LIN {X 0,Y 284.606,Z 589.036,A -85,B 0,C 180,E1 -17094.331,E2 -17094.331} C_VEL
LIN {X 0,Y 284.86,Z 589.002,A -85,B 0,C 180,E1 -17098.586,E2 -17098.586} C_VEL
LIN {X 0,Y 284.86,Z 588.997,A -85,B 0,C 180,E1 -17101.413,E2 -17101.413} C_VEL
LIN {X 0,Y 284.703,Z 589.017,A -85,B 0,C 180,E1 -17107.089,E2 -17107.089} C_VEL
LIN {X 0,Y 284.571,Z 589.036,A -85,B 0,C 180,E1 -17109.955,E2 -17109.955} C_VEL
LIN {X 0,Y 284.482,Z 589.046,A -85,B 0,C 180,E1 -17114.302,E2 -17114.302} C_VEL
LIN {X 0,Y 284.429,Z 589.048,A -85,B 0,C 180,E1 -17117.247,E2 -17117.247} C_VEL
LIN {X 0,Y 284.382,Z 589.061,A -85,B 0,C 180,E1 -17120.241,E2 -17120.241} C_VEL
LIN {X 0,Y 284.372,Z 589.06,A -85,B 0,C 180,E1 -17123.874,E2 -17123.874} C_VEL
LIN {X 0,Y 284.4,Z 589.052,A -85,B 0,C 180,E1 -17127.173,E2 -17127.173} C_VEL
LIN {X 0,Y 284.298,Z 589.069,A -85,B 0,C 180,E1 -17131.273,E2 -17131.273} C_VEL
LIN {X 0,Y 284.343,Z 589.063,A -85,B 0,C 180,E1 -17135.347,E2 -17135.347} C_VEL
LIN {X 0,Y 284.314,Z 589.069,A -85,B 0,C 180,E1 -17138.168,E2 -17138.168} C_VEL
LIN {X 0,Y 284.271,Z 589.074,A -85,B 0,C 180,E1 -17142.123,E2 -17142.123} C_VEL
LIN {X 0,Y 284.287,Z 589.069,A -85,B 0,C 180,E1 -17146.194,E2 -17146.194} C_VEL
LIN {X 0,Y 284.314,Z 589.068,A -85,B 0,C 180,E1 -17150.021,E2 -17150.021} C_VEL
LIN {X 0,Y 284.351,Z 589.061,A -85,B 0,C 180,E1 -17153.616,E2 -17153.616} C_VEL
LIN {X 0,Y 284.308,Z 589.067,A -85,B 0,C 180,E1 -17157.189,E2 -17157.189} C_VEL
LIN {X 0,Y 284.356,Z 589.065,A -85,B 0,C 180,E1 -17160.374,E2 -17160.374} C_VEL
LIN {X 0,Y 284.375,Z 589.058,A -85,B 0,C 180,E1 -17163.585,E2 -17163.585} C_VEL
LIN {X 0,Y 284.367,Z 589.063,A -85,B 0,C 180,E1 -17166.706,E2 -17166.706} C_VEL
LIN {X 0,Y 284.403,Z 589.057,A -85,B 0,C 180,E1 -17171.26,E2 -17171.26} C_VEL
LIN {X 0,Y 284.492,Z 589.045,A -85,B 0,C 180,E1 -17174.458,E2 -17174.458} C_VEL
LIN {X 0,Y 284.489,Z 589.047,A -85,B 0,C 180,E1 -17178.6,E2 -17178.6} C_VEL
LIN {X 0,Y 284.668,Z 589.024,A -85,B 0,C 180,E1 -17181.525,E2 -17181.525} C_VEL
LIN {X 0,Y 288.557,Z 601.326,A -85,B 0,C 180,E1 -17182.828,E2 -17182.828} C_VEL
LIN {X 0,Y 291.525,Z 612.433,A -85,B 0,C 180,E1 -17184.223,E2 -17184.223} C_VEL
LIN {X 0,Y 291.996,Z 614.209,A -85,B 0,C 180,E1 -17184.474,E2 -17184.474} C_VEL
LIN {X 0,Y 290.847,Z 625.708,A -85,B 0,C 180,E1 -17186.015,E2 -17186.015} C_VEL
LIN {X 0,Y 289.812,Z 634.995,A -85,B 0,C 180,E1 -17187.567,E2 -17187.567} C_VEL
LIN {X 0,Y 288.604,Z 643.761,A -85,B 0,C 180,E1 -17189.353,E2 -17189.353} C_VEL
LIN {X 0,Y 287.536,Z 651.804,A -85,B 0,C 180,E1 -17191.399,E2 -17191.399} C_VEL
LIN {X 0,Y 286.639,Z 658.483,A -85,B 0,C 180,E1 -17193.513,E2 -17193.513} C_VEL
LIN {X 0,Y 285.832,Z 663.856,A -85,B 0,C 180,E1 -17195.643,E2 -17195.643} C_VEL
LIN {X 0,Y 285.275,Z 668.057,A -85,B 0,C 180,E1 -17197.786,E2 -17197.786} C_VEL
LIN {X 0,Y 284.872,Z 671.215,A -85,B 0,C 180,E1 -17199.943,E2 -17199.943} C_VEL
LIN {X 0,Y 284.756,Z 672.789,A -85,B 0,C 180,E1 -17201.386,E2 -17201.386} C_VEL
LIN {X 0,Y 284.704,Z 673.91,A -85,B 0,C 180,E1 -17202.835,E2 -17202.835} C_VEL
LIN {X 0,Y 284.97,Z 674.965,A -85,B 0,C 180,E1 -17205.739,E2 -17205.739} C_VEL
LIN {X 0,Y 285.182,Z 674.889,A -85,B 0,C 180,E1 -17207.2,E2 -17207.2} C_VEL
LIN {X 0,Y 285.511,Z 674.378,A -85,B 0,C 180,E1 -17208.661,E2 -17208.661} C_VEL
LIN {X 0,Y 286.381,Z 672.543,A -85,B 0,C 180,E1 -17211.166,E2 -17211.166} C_VEL
LIN {X 0,Y 287.626,Z 669.263,A -85,B 0,C 180,E1 -17213.775,E2 -17213.775} C_VEL
LIN {X 0,Y 288.934,Z 665.274,A -85,B 0,C 180,E1 -17215.964,E2 -17215.964} C_VEL
LIN {X 0,Y 290.739,Z 659.013,A -85,B 0,C 180,E1 -17218.515,E2 -17218.515} C_VEL
LIN {X 0,Y 292.655,Z 652.073,A -85,B 0,C 180,E1 -17220.683,E2 -17220.683} C_VEL
LIN {X 0,Y 294.442,Z 644.856,A -85,B 0,C 180,E1 -17222.481,E2 -17222.481} C_VEL
LIN {X 0,Y 296.435,Z 635.72,A -85,B 0,C 180,E1 -17224.316,E2 -17224.316} C_VEL
LIN {X 0,Y 298.194,Z 626.062,A -85,B 0,C 180,E1 -17225.889,E2 -17225.889} C_VEL
LIN {X 0,Y 295.848,Z 617.051,A -85,B 0,C 180,E1 -17227.55,E2 -17227.55} C_VEL
LIN {X 0,Y 291.54,Z 610.398,A -85,B 0,C 180,E1 -17228.962,E2 -17228.962} C_VEL
LIN {X 0,Y 287.015,Z 604.55,A -85,B 0,C 180,E1 -17230.228,E2 -17230.228} C_VEL
LIN {X 0,Y 286.747,Z 603.732,A -85,B 0,C 180,E1 -17230.381,E2 -17230.381} C_VEL
LIN {X 0,Y 286.527,Z 609.898,A -85,B 0,C 180,E1 -17233.374,E2 -17233.374} C_VEL
LIN {X 0,Y 285.989,Z 617.64,A -85,B 0,C 180,E1 -17237.095,E2 -17237.095} C_VEL
LIN {X 0,Y 285.473,Z 626.048,A -85,B 0,C 180,E1 -17241.114,E2 -17241.114} C_VEL
LIN {X 0,Y 285.15,Z 632.582,A -85,B 0,C 180,E1 -17244.221,E2 -17244.221} C_VEL
LIN {X 0,Y 287.62,Z 646.522,A -85,B 0,C 180,E1 -17245.077,E2 -17245.077} C_VEL
LIN {X 0,Y 289.828,Z 659.569,A -85,B 0,C 180,E1 -17246.148,E2 -17246.148} C_VEL
LIN {X 0,Y 290.365,Z 664.219,A -85,B 0,C 180,E1 -17246.59,E2 -17246.59} C_VEL
LIN {X 0,Y 289.25,Z 676.311,A -85,B 0,C 180,E1 -17247.822,E2 -17247.822} C_VEL
LIN {X 0,Y 287.885,Z 688.211,A -85,B 0,C 180,E1 -17249.363,E2 -17249.363} C_VEL
LIN {X 0,Y 286.677,Z 698.653,A -85,B 0,C 180,E1 -17251.042,E2 -17251.042} C_VEL
LIN {X 0,Y 285.548,Z 708.096,A -85,B 0,C 180,E1 -17252.915,E2 -17252.915} C_VEL
LIN {X 0,Y 284.575,Z 715.877,A -85,B 0,C 180,E1 -17254.786,E2 -17254.786} C_VEL
LIN {X 0,Y 283.779,Z 723.483,A -85,B 0,C 180,E1 -17257.042,E2 -17257.042} C_VEL
LIN {X 0,Y 283.086,Z 730.338,A -85,B 0,C 180,E1 -17259.662,E2 -17259.662} C_VEL
LIN {X 0,Y 282.716,Z 734.782,A -85,B 0,C 180,E1 -17261.897,E2 -17261.897} C_VEL
LIN {X 0,Y 282.461,Z 738.031,A -85,B 0,C 180,E1 -17264.116,E2 -17264.116} C_VEL
LIN {X 0,Y 282.44,Z 739.964,A -85,B 0,C 180,E1 -17266.028,E2 -17266.028} C_VEL
LIN {X 0,Y 282.528,Z 741.392,A -85,B 0,C 180,E1 -17268.522,E2 -17268.522} C_VEL
LIN {X 0,Y 282.699,Z 741.622,A -85,B 0,C 180,E1 -17269.979,E2 -17269.979} C_VEL
LIN {X 0,Y 283.343,Z 740.915,A -85,B 0,C 180,E1 -17272.804,E2 -17272.804} C_VEL
LIN {X 0,Y 283.79,Z 739.87,A -85,B 0,C 180,E1 -17274.316,E2 -17274.316} C_VEL
LIN {X 0,Y 284.213,Z 738.56,A -85,B 0,C 180,E1 -17275.642,E2 -17275.642} C_VEL
LIN {X 0,Y 284.048,Z 737.349,A -85,B 0,C 180,E1 -17276.809,E2 -17276.809} C_VEL
LIN {X 0,Y 282.237,Z 735.003,A -85,B 0,C 180,E1 -17278.726,E2 -17278.726} C_VEL
LIN {X 0,Y 280.85,Z 732.632,A -85,B 0,C 180,E1 -17280.244,E2 -17280.244} C_VEL
LIN {X 0,Y 280.68,Z 730.45,A -85,B 0,C 180,E1 -17281.364,E2 -17281.364} C_VEL
LIN {X 0,Y 280.899,Z 729.624,A -85,B 0,C 180,E1 -17281.727,E2 -17281.727} C_VEL
LIN {X 0,Y 282.965,Z 723.832,A -85,B 0,C 180,E1 -17283.917,E2 -17283.917} C_VEL
LIN {X 0,Y 285.304,Z 716.83,A -85,B 0,C 180,E1 -17286.01,E2 -17286.01} C_VEL
LIN {X 0,Y 288.012,Z 708.164,A -85,B 0,C 180,E1 -17288.066,E2 -17288.066} C_VEL
LIN {X 0,Y 290.524,Z 699.534,A -85,B 0,C 180,E1 -17289.75,E2 -17289.75} C_VEL
LIN {X 0,Y 293.371,Z 688.781,A -85,B 0,C 180,E1 -17291.434,E2 -17291.434} C_VEL
LIN {X 0,Y 295.827,Z 677.662,A -85,B 0,C 180,E1 -17292.845,E2 -17292.845} C_VEL
LIN {X 0,Y 294.677,Z 667.632,A -85,B 0,C 180,E1 -17294.47,E2 -17294.47} C_VEL
LIN {X 0,Y 292.135,Z 657.124,A -85,B 0,C 180,E1 -17296.234,E2 -17296.234} C_VEL
LIN {X 0,Y 288.644,Z 647.19,A -85,B 0,C 180,E1 -17298.026,E2 -17298.026} C_VEL
LIN {X 0,Y 286.586,Z 642.357,A -85,B 0,C 180,E1 -17298.985,E2 -17298.985} C_VEL
LIN {X 0,Y 285.531,Z 639.392,A -85,B 0,C 180,E1 -17299.548,E2 -17299.548} C_VEL
LIN {X 0,Y 287.353,Z 632.653,A -85,B 0,C 180,E1 -17303.801,E2 -17303.801} C_VEL
LIN {X 0,Y 288.082,Z 629.504,A -85,B 0,C 180,E1 -17306.049,E2 -17306.049} C_VEL
LIN {X 0,Y 288.296,Z 626.554,A -85,B 0,C 180,E1 -17308.65,E2 -17308.65} C_VEL
LIN {X 0,Y 288.285,Z 624.039,A -85,B 0,C 180,E1 -17311.436,E2 -17311.436} C_VEL
LIN {X 0,Y 288.31,Z 622.174,A -85,B 0,C 180,E1 -17314.102,E2 -17314.102} C_VEL
LIN {X 0,Y 288.543,Z 620.675,A -85,B 0,C 180,E1 -17317.512,E2 -17317.512} C_VEL
LIN {X 0,Y 288.683,Z 620.382,A -85,B 0,C 180,E1 -17319.27,E2 -17319.27} C_VEL
LIN {X 0,Y 288.734,Z 620.549,A -85,B 0,C 180,E1 -17321.087,E2 -17321.087} C_VEL
LIN {X 0,Y 288.549,Z 621.433,A -85,B 0,C 180,E1 -17323.058,E2 -17323.058} C_VEL
LIN {X 0,Y 288.243,Z 623.559,A -85,B 0,C 180,E1 -17325.684,E2 -17325.684} C_VEL
LIN {X 0,Y 288.344,Z 627.834,A -85,B 0,C 180,E1 -17329.077,E2 -17329.077} C_VEL
LIN {X 0,Y 288.366,Z 629.026,A -85,B 0,C 180,E1 -17329.796,E2 -17329.796} C_VEL
LIN {X 0,Y 287.752,Z 633.355,A -85,B 0,C 180,E1 -17331.717,E2 -17331.717} C_VEL
LIN {X 0,Y 286.85,Z 639.765,A -85,B 0,C 180,E1 -17333.986,E2 -17333.986} C_VEL
LIN {X 0,Y 286.34,Z 648.27,A -85,B 0,C 180,E1 -17336.565,E2 -17336.565} C_VEL
LIN {X 0,Y 286.351,Z 652.539,A -85,B 0,C 180,E1 -17337.652,E2 -17337.652} C_VEL
LIN {X 0,Y 289.68,Z 665.175,A -85,B 0,C 180,E1 -17339.394,E2 -17339.394} C_VEL
LIN {X 0,Y 291.628,Z 675.536,A -85,B 0,C 180,E1 -17340.711,E2 -17340.711} C_VEL
LIN {X 0,Y 292.656,Z 687.693,A -85,B 0,C 180,E1 -17342.173,E2 -17342.173} C_VEL
LIN {X 0,Y 292.149,Z 698.271,A -85,B 0,C 180,E1 -17343.413,E2 -17343.413} C_VEL
LIN {X 0,Y 290.389,Z 710.468,A -85,B 0,C 180,E1 -17344.944,E2 -17344.944} C_VEL
LIN {X 0,Y 288.295,Z 721.832,A -85,B 0,C 180,E1 -17346.665,E2 -17346.665} C_VEL
LIN {X 0,Y 285.663,Z 731.527,A -85,B 0,C 180,E1 -17348.345,E2 -17348.345} C_VEL
LIN {X 0,Y 283.312,Z 739.677,A -85,B 0,C 180,E1 -17350.058,E2 -17350.058} C_VEL
LIN {X 0,Y 280.506,Z 749.053,A -85,B 0,C 180,E1 -17352.504,E2 -17352.504} C_VEL
LIN {X 0,Y 278.866,Z 755.583,A -85,B 0,C 180,E1 -17354.657,E2 -17354.657} C_VEL
LIN {X 0,Y 277.3,Z 760.909,A -85,B 0,C 180,E1 -17356.816,E2 -17356.816} C_VEL
LIN {X 0,Y 276.397,Z 765.123,A -85,B 0,C 180,E1 -17359.008,E2 -17359.008} C_VEL
LIN {X 0,Y 275.824,Z 768.335,A -85,B 0,C 180,E1 -17361.208,E2 -17361.208} C_VEL
LIN {X 0,Y 275.613,Z 769.942,A -85,B 0,C 180,E1 -17362.676,E2 -17362.676} C_VEL
LIN {X 0,Y 275.476,Z 771.938,A -85,B 0,C 180,E1 -17365.612,E2 -17365.612} C_VEL
LIN {X 0,Y 275.507,Z 772.333,A -85,B 0,C 180,E1 -17367.077,E2 -17367.077} C_VEL
LIN {X 0,Y 275.887,Z 771.819,A -85,B 0,C 180,E1 -17370.001,E2 -17370.001} C_VEL
LIN {X 0,Y 275.746,Z 770.912,A -85,B 0,C 180,E1 -17371.462,E2 -17371.462} C_VEL
LIN {X 0,Y 275.594,Z 769.545,A -85,B 0,C 180,E1 -17372.925,E2 -17372.925} C_VEL
LIN {X 0,Y 275.671,Z 766.636,A -85,B 0,C 180,E1 -17375.121,E2 -17375.121} C_VEL
LIN {X 0,Y 275.725,Z 762.583,A -85,B 0,C 180,E1 -17377.323,E2 -17377.323} C_VEL
LIN {X 0,Y 276.04,Z 756.286,A -85,B 0,C 180,E1 -17379.897,E2 -17379.897} C_VEL
LIN {X 0,Y 276.598,Z 749.373,A -85,B 0,C 180,E1 -17382.101,E2 -17382.101} C_VEL
LIN {X 0,Y 277.519,Z 740.696,A -85,B 0,C 180,E1 -17384.296,E2 -17384.296} C_VEL
LIN {X 0,Y 278.308,Z 733.752,A -85,B 0,C 180,E1 -17385.753,E2 -17385.753} C_VEL
LIN {X 0,Y 279.563,Z 723.375,A -85,B 0,C 180,E1 -17387.559,E2 -17387.559} C_VEL
LIN {X 0,Y 280.95,Z 711.747,A -85,B 0,C 180,E1 -17389.168,E2 -17389.168} C_VEL
LIN {X 0,Y 281.033,Z 701.802,A -85,B 0,C 180,E1 -17390.304,E2 -17390.304} C_VEL
LIN {X 0,Y 280.708,Z 689.594,A -85,B 0,C 180,E1 -17391.437,E2 -17391.437} C_VEL
LIN {X 0,Y 279.865,Z 675.724,A -85,B 0,C 180,E1 -17392.421,E2 -17392.421} C_VEL
LIN {X 0,Y 278.595,Z 659.43,A -85,B 0,C 180,E1 -17393.609,E2 -17393.609} C_VEL
LIN {X 0,Y 277.646,Z 651.097,A -85,B 0,C 180,E1 -17394.076,E2 -17394.076} C_VEL
LIN {X 0,Y 277.221,Z 642.295,A -85,B 0,C 180,E1 -17395.156,E2 -17395.156} C_VEL
LIN {X 0,Y 278.337,Z 631.986,A -85,B 0,C 180,E1 -17399.498,E2 -17399.498} C_VEL
LIN {X 0,Y 279.78,Z 621.349,A -85,B 0,C 180,E1 -17404.008,E2 -17404.008} C_VEL
LIN {X 0,Y 281.164,Z 612.603,A -85,B 0,C 180,E1 -17407.765,E2 -17407.765} C_VEL
LIN {X 0,Y 281.019,Z 609.529,A -85,B 0,C 180,E1 -17409.169,E2 -17409.169} C_VEL
LIN {X 0,Y 279.688,Z 602.149,A -85,B 0,C 180,E1 -17412.724,E2 -17412.724} C_VEL
LIN {X 0,Y 277.98,Z 593.465,A -85,B 0,C 180,E1 -17417.156,E2 -17417.156} C_VEL
LIN {X 0,Y 277.252,Z 589.953,A -85,B 0,C 180,E1 -17419.092,E2 -17419.092} C_VEL
LIN {X 0,Y 277.287,Z 589.951,A -85,B 0,C 180,E1 -17422.533,E2 -17422.533} C_VEL
LIN {X 0,Y 277.26,Z 589.953,A -85,B 0,C 180,E1 -17426.105,E2 -17426.105} C_VEL
LIN {X 0,Y 277.267,Z 589.947,A -85,B 0,C 180,E1 -17429.539,E2 -17429.539} C_VEL
LIN {X 0,Y 277.363,Z 589.934,A -85,B 0,C 180,E1 -17432.864,E2 -17432.864} C_VEL
LIN {X 0,Y 277.334,Z 589.94,A -85,B 0,C 180,E1 -17436.079,E2 -17436.079} C_VEL
LIN {X 0,Y 277.35,Z 589.937,A -85,B 0,C 180,E1 -17440.766,E2 -17440.766} C_VEL
LIN {X 0,Y 277.44,Z 589.925,A -85,B 0,C 180,E1 -17445.326,E2 -17445.326} C_VEL
LIN {X 0,Y 277.512,Z 589.916,A -85,B 0,C 180,E1 -17449.788,E2 -17449.788} C_VEL
LIN {X 0,Y 277.659,Z 589.898,A -85,B 0,C 180,E1 -17452.729,E2 -17452.729} C_VEL
LIN {X 0,Y 277.826,Z 589.879,A -85,B 0,C 180,E1 -17458.55,E2 -17458.55} C_VEL
LIN {X 0,Y 277.826,Z 589.874,A -85,B 0,C 180,E1 -17461.449,E2 -17461.449} C_VEL
LIN {X 0,Y 277.658,Z 589.894,A -85,B 0,C 180,E1 -17467.27,E2 -17467.27} C_VEL
LIN {X 0,Y 277.511,Z 589.917,A -85,B 0,C 180,E1 -17470.211,E2 -17470.211} C_VEL
LIN {X 0,Y 277.432,Z 589.92,A -85,B 0,C 180,E1 -17474.674,E2 -17474.674} C_VEL
LIN {X 0,Y 277.349,Z 589.934,A -85,B 0,C 180,E1 -17479.233,E2 -17479.233} C_VEL
LIN {X 0,Y 277.323,Z 589.94,A -85,B 0,C 180,E1 -17484.169,E2 -17484.169} C_VEL
LIN {X 0,Y 277.329,Z 589.932,A -85,B 0,C 180,E1 -17487.504,E2 -17487.504} C_VEL
LIN {X 0,Y 277.275,Z 589.948,A -85,B 0,C 180,E1 -17490.48,E2 -17490.48} C_VEL
LIN {X 0,Y 277.25,Z 589.947,A -85,B 0,C 180,E1 -17493.895,E2 -17493.895} C_VEL
LIN {X 0,Y 277.27,Z 589.944,A -85,B 0,C 180,E1 -17497.468,E2 -17497.468} C_VEL
LIN {X 0,Y 277.212,Z 589.952,A -85,B 0,C 180,E1 -17501.235,E2 -17501.235} C_VEL
LIN {X 0,Y 277.224,Z 589.946,A -85,B 0,C 180,E1 -17505.221,E2 -17505.221} C_VEL
LIN {X 0,Y 277.228,Z 589.952,A -85,B 0,C 180,E1 -17508.765,E2 -17508.765} C_VEL
LIN {X 0,Y 277.283,Z 589.943,A -85,B 0,C 180,E1 -17512.532,E2 -17512.532} C_VEL
LIN {X 0,Y 277.255,Z 589.948,A -85,B 0,C 180,E1 -17516.104,E2 -17516.104} C_VEL
LIN {X 0,Y 277.262,Z 589.945,A -85,B 0,C 180,E1 -17519.537,E2 -17519.537} C_VEL
LIN {X 0,Y 277.356,Z 589.934,A -85,B 0,C 180,E1 -17522.863,E2 -17522.863} C_VEL
LIN {X 0,Y 277.329,Z 589.939,A -85,B 0,C 180,E1 -17526.078,E2 -17526.078} C_VEL
LIN {X 0,Y 277.345,Z 589.939,A -85,B 0,C 180,E1 -17530.765,E2 -17530.765} C_VEL
LIN {X 0,Y 277.435,Z 589.924,A -85,B 0,C 180,E1 -17535.325,E2 -17535.325} C_VEL
LIN {X 0,Y 277.507,Z 589.917,A -85,B 0,C 180,E1 -17539.787,E2 -17539.787} C_VEL
LIN {X 0,Y 277.617,Z 589.902,A -85,B 0,C 180,E1 -17541.053,E2 -17541.053} C_VEL
LIN {X 0,Y 281.357,Z 601.323,A -85,B 0,C 180,E1 -17542.283,E2 -17542.283} C_VEL
LIN {X 0,Y 284.209,Z 612.288,A -85,B 0,C 180,E1 -17543.672,E2 -17543.672} C_VEL
LIN {X 0,Y 285.038,Z 615.32,A -85,B 0,C 180,E1 -17544.107,E2 -17544.107} C_VEL
LIN {X 0,Y 284.246,Z 624.779,A -85,B 0,C 180,E1 -17545.39,E2 -17545.39} C_VEL
LIN {X 0,Y 283.02,Z 635.357,A -85,B 0,C 180,E1 -17547.152,E2 -17547.152} C_VEL
LIN {X 0,Y 281.727,Z 644.666,A -85,B 0,C 180,E1 -17549.076,E2 -17549.076} C_VEL
LIN {X 0,Y 280.649,Z 652.285,A -85,B 0,C 180,E1 -17551.039,E2 -17551.039} C_VEL
LIN {X 0,Y 279.701,Z 659.158,A -85,B 0,C 180,E1 -17553.24,E2 -17553.24} C_VEL
LIN {X 0,Y 278.75,Z 665.41,A -85,B 0,C 180,E1 -17555.787,E2 -17555.787} C_VEL
LIN {X 0,Y 278.187,Z 669.492,A -85,B 0,C 180,E1 -17557.986,E2 -17557.986} C_VEL
LIN {X 0,Y 277.805,Z 672.538,A -85,B 0,C 180,E1 -17560.199,E2 -17560.199} C_VEL
LIN {X 0,Y 277.702,Z 674.009,A -85,B 0,C 180,E1 -17561.679,E2 -17561.679} C_VEL
LIN {X 0,Y 277.778,Z 675.743,A -85,B 0,C 180,E1 -17564.654,E2 -17564.654} C_VEL
LIN {X 0,Y 278.023,Z 676.005,A -85,B 0,C 180,E1 -17566.143,E2 -17566.143} C_VEL
LIN {X 0,Y 278.26,Z 675.84,A -85,B 0,C 180,E1 -17567.641,E2 -17567.641} C_VEL
LIN {X 0,Y 278.625,Z 675.278,A -85,B 0,C 180,E1 -17569.14,E2 -17569.14} C_VEL
LIN {X 0,Y 279.528,Z 673.5,A -85,B 0,C 180,E1 -17571.525,E2 -17571.525} C_VEL
LIN {X 0,Y 280.932,Z 669.885,A -85,B 0,C 180,E1 -17574.378,E2 -17574.378} C_VEL
LIN {X 0,Y 282.345,Z 665.765,A -85,B 0,C 180,E1 -17576.617,E2 -17576.617} C_VEL
LIN {X 0,Y 283.998,Z 660.378,A -85,B 0,C 180,E1 -17578.851,E2 -17578.851} C_VEL
LIN {X 0,Y 285.99,Z 653.521,A -85,B 0,C 180,E1 -17581.066,E2 -17581.066} C_VEL
LIN {X 0,Y 287.84,Z 646.411,A -85,B 0,C 180,E1 -17582.904,E2 -17582.904} C_VEL
LIN {X 0,Y 290.079,Z 636.717,A -85,B 0,C 180,E1 -17584.903,E2 -17584.903} C_VEL
LIN {X 0,Y 291.669,Z 628.681,A -85,B 0,C 180,E1 -17586.255,E2 -17586.255} C_VEL
LIN {X 0,Y 290.789,Z 623.926,A -85,B 0,C 180,E1 -17587.171,E2 -17587.171} C_VEL
LIN {X 0,Y 289.625,Z 620.101,A -85,B 0,C 180,E1 -17587.916,E2 -17587.916} C_VEL
LIN {X 0,Y 283.77,Z 611.791,A -85,B 0,C 180,E1 -17589.848,E2 -17589.848} C_VEL
LIN {X 0,Y 281.937,Z 609.423,A -85,B 0,C 180,E1 -17590.398,E2 -17590.398} C_VEL
LIN {X 0,Y 280.676,Z 608.353,A -85,B 0,C 180,E1 -17590.705,E2 -17590.705} C_VEL
LIN {X 0,Y 279.77,Z 606.539,A -85,B 0,C 180,E1 -17591.053,E2 -17591.053} C_VEL
LIN {X 0,Y 279.341,Z 614.142,A -85,B 0,C 180,E1 -17594.783,E2 -17594.783} C_VEL
LIN {X 0,Y 278.695,Z 623.179,A -85,B 0,C 180,E1 -17599.156,E2 -17599.156} C_VEL
LIN {X 0,Y 278.195,Z 631.942,A -85,B 0,C 180,E1 -17603.384,E2 -17603.384} C_VEL
LIN {X 0,Y 278.193,Z 633.111,A -85,B 0,C 180,E1 -17603.877,E2 -17603.877} C_VEL
LIN {X 0,Y 280.679,Z 647.191,A -85,B 0,C 180,E1 -17604.772,E2 -17604.772} C_VEL
LIN {X 0,Y 283,Z 661.237,A -85,B 0,C 180,E1 -17605.974,E2 -17605.974} C_VEL
LIN {X 0,Y 283.378,Z 665.151,A -85,B 0,C 180,E1 -17606.362,E2 -17606.362} C_VEL
LIN {X 0,Y 282.29,Z 676.434,A -85,B 0,C 180,E1 -17607.543,E2 -17607.543} C_VEL
LIN {X 0,Y 280.872,Z 688.513,A -85,B 0,C 180,E1 -17609.14,E2 -17609.14} C_VEL
LIN {X 0,Y 279.66,Z 698.989,A -85,B 0,C 180,E1 -17610.863,E2 -17610.863} C_VEL
LIN {X 0,Y 278.395,Z 709.305,A -85,B 0,C 180,E1 -17612.974,E2 -17612.974} C_VEL
LIN {X 0,Y 277.403,Z 717.108,A -85,B 0,C 180,E1 -17614.931,E2 -17614.931} C_VEL
LIN {X 0,Y 276.639,Z 724.416,A -85,B 0,C 180,E1 -17617.206,E2 -17617.206} C_VEL
LIN {X 0,Y 276.094,Z 729.425,A -85,B 0,C 180,E1 -17619.123,E2 -17619.123} C_VEL
LIN {X 0,Y 275.676,Z 734.164,A -85,B 0,C 180,E1 -17621.418,E2 -17621.418} C_VEL
LIN {X 0,Y 275.389,Z 737.699,A -85,B 0,C 180,E1 -17623.697,E2 -17623.697} C_VEL
LIN {X 0,Y 275.34,Z 740.106,A -85,B 0,C 180,E1 -17625.909,E2 -17625.909} C_VEL
LIN {X 0,Y 275.43,Z 741.605,A -85,B 0,C 180,E1 -17628.222,E2 -17628.222} C_VEL
LIN {X 0,Y 275.579,Z 742.047,A -85,B 0,C 180,E1 -17629.717,E2 -17629.717} C_VEL
LIN {X 0,Y 275.84,Z 742.055,A -85,B 0,C 180,E1 -17631.207,E2 -17631.207} C_VEL
LIN {X 0,Y 276.262,Z 741.57,A -85,B 0,C 180,E1 -17632.799,E2 -17632.799} C_VEL
LIN {X 0,Y 277.151,Z 739.605,A -85,B 0,C 180,E1 -17635.638,E2 -17635.638} C_VEL
LIN {X 0,Y 278.187,Z 736.982,A -85,B 0,C 180,E1 -17637.829,E2 -17637.829} C_VEL
LIN {X 0,Y 279.584,Z 733.346,A -85,B 0,C 180,E1 -17640.001,E2 -17640.001} C_VEL
LIN {X 0,Y 280.899,Z 729.624,A -85,B 0,C 180,E1 -17641.727,E2 -17641.727} C_VEL
LIN {X 0,Y 281.22,Z 727.146,A -85,B 0,C 180,E1 -17642.818,E2 -17642.818} C_VEL
LIN {X 0,Y 280.234,Z 722.98,A -85,B 0,C 180,E1 -17644.645,E2 -17644.645} C_VEL
LIN {X 0,Y 279.421,Z 718.315,A -85,B 0,C 180,E1 -17646.423,E2 -17646.423} C_VEL
LIN {X 0,Y 279.987,Z 714.995,A -85,B 0,C 180,E1 -17647.416,E2 -17647.416} C_VEL
LIN {X 0,Y 282.736,Z 706.842,A -85,B 0,C 180,E1 -17649.299,E2 -17649.299} C_VEL
LIN {X 0,Y 285.773,Z 696.756,A -85,B 0,C 180,E1 -17651.168,E2 -17651.168} C_VEL
LIN {X 0,Y 288.783,Z 685.636,A -85,B 0,C 180,E1 -17652.831,E2 -17652.831} C_VEL
LIN {X 0,Y 290.04,Z 680.443,A -85,B 0,C 180,E1 -17653.488,E2 -17653.488} C_VEL
LIN {X 0,Y 289.609,Z 673.403,A -85,B 0,C 180,E1 -17654.675,E2 -17654.675} C_VEL
LIN {X 0,Y 287.785,Z 663.263,A -85,B 0,C 180,E1 -17656.476,E2 -17656.476} C_VEL
LIN {X 0,Y 284.849,Z 653.325,A -85,B 0,C 180,E1 -17658.363,E2 -17658.363} C_VEL
LIN {X 0,Y 281.173,Z 643.852,A -85,B 0,C 180,E1 -17660.34,E2 -17660.34} C_VEL
LIN {X 0,Y 279.742,Z 640.057,A -85,B 0,C 180,E1 -17661.202,E2 -17661.202} C_VEL
LIN {X 0,Y 281.22,Z 635.336,A -85,B 0,C 180,E1 -17664.353,E2 -17664.353} C_VEL
LIN {X 0,Y 281.957,Z 632.366,A -85,B 0,C 180,E1 -17666.659,E2 -17666.659} C_VEL
LIN {X 0,Y 282.19,Z 629.601,A -85,B 0,C 180,E1 -17669.349,E2 -17669.349} C_VEL
LIN {X 0,Y 282.302,Z 627.32,A -85,B 0,C 180,E1 -17672.177,E2 -17672.177} C_VEL
LIN {X 0,Y 282.456,Z 625.761,A -85,B 0,C 180,E1 -17674.91,E2 -17674.91} C_VEL
LIN {X 0,Y 282.727,Z 624.862,A -85,B 0,C 180,E1 -17677.305,E2 -17677.305} C_VEL
LIN {X 0,Y 282.969,Z 624.61,A -85,B 0,C 180,E1 -17679.655,E2 -17679.655} C_VEL
LIN {X 0,Y 282.945,Z 625.292,A -85,B 0,C 180,E1 -17682.118,E2 -17682.118} C_VEL
LIN {X 0,Y 282.746,Z 626.648,A -85,B 0,C 180,E1 -17684.106,E2 -17684.106} C_VEL
LIN {X 0,Y 282.681,Z 629.477,A -85,B 0,C 180,E1 -17686.868,E2 -17686.868} C_VEL
LIN {X 0,Y 282.836,Z 632.31,A -85,B 0,C 180,E1 -17688.958,E2 -17688.958} C_VEL
LIN {X 0,Y 282.542,Z 635.249,A -85,B 0,C 180,E1 -17690.453,E2 -17690.453} C_VEL
LIN {X 0,Y 281.567,Z 641.182,A -85,B 0,C 180,E1 -17692.753,E2 -17692.753} C_VEL
LIN {X 0,Y 280.724,Z 650.383,A -85,B 0,C 180,E1 -17695.707,E2 -17695.707} C_VEL
LIN {X 0,Y 280.726,Z 652.091,A -85,B 0,C 180,E1 -17696.127,E2 -17696.127} C_VEL
LIN {X 0,Y 283.994,Z 664.357,A -85,B 0,C 180,E1 -17698.025,E2 -17698.025} C_VEL
LIN {X 0,Y 286.302,Z 677.17,A -85,B 0,C 180,E1 -17699.782,E2 -17699.782} C_VEL
LIN {X 0,Y 287.029,Z 689.116,A -85,B 0,C 180,E1 -17701.324,E2 -17701.324} C_VEL
LIN {X 0,Y 286.589,Z 697.866,A -85,B 0,C 180,E1 -17702.414,E2 -17702.414} C_VEL
LIN {X 0,Y 284.644,Z 710.053,A -85,B 0,C 180,E1 -17704.009,E2 -17704.009} C_VEL
LIN {X 0,Y 282.211,Z 722.401,A -85,B 0,C 180,E1 -17705.935,E2 -17705.935} C_VEL
LIN {X 0,Y 279.159,Z 732.656,A -85,B 0,C 180,E1 -17707.814,E2 -17707.814} C_VEL
LIN {X 0,Y 276.234,Z 741.938,A -85,B 0,C 180,E1 -17709.913,E2 -17709.913} C_VEL
LIN {X 0,Y 273.757,Z 749.612,A -85,B 0,C 180,E1 -17712.059,E2 -17712.059} C_VEL
LIN {X 0,Y 272.01,Z 755.894,A -85,B 0,C 180,E1 -17714.26,E2 -17714.26} C_VEL
LIN {X 0,Y 270.383,Z 761.02,A -85,B 0,C 180,E1 -17716.473,E2 -17716.473} C_VEL
LIN {X 0,Y 269.391,Z 765.1,A -85,B 0,C 180,E1 -17718.718,E2 -17718.718} C_VEL
LIN {X 0,Y 268.768,Z 768.19,A -85,B 0,C 180,E1 -17720.975,E2 -17720.975} C_VEL
LIN {X 0,Y 268.402,Z 770.842,A -85,B 0,C 180,E1 -17723.989,E2 -17723.989} C_VEL
LIN {X 0,Y 268.378,Z 771.582,A -85,B 0,C 180,E1 -17725.496,E2 -17725.496} C_VEL
LIN {X 0,Y 268.43,Z 771.872,A -85,B 0,C 180,E1 -17727,E2 -17727} C_VEL
LIN {X 0,Y 268.828,Z 771.238,A -85,B 0,C 180,E1 -17730.001,E2 -17730.001} C_VEL
LIN {X 0,Y 268.658,Z 770.26,A -85,B 0,C 180,E1 -17731.5,E2 -17731.5} C_VEL
LIN {X 0,Y 268.521,Z 768.797,A -85,B 0,C 180,E1 -17733.002,E2 -17733.002} C_VEL
LIN {X 0,Y 268.596,Z 765.282,A -85,B 0,C 180,E1 -17735.566,E2 -17735.566} C_VEL
LIN {X 0,Y 268.717,Z 759.978,A -85,B 0,C 180,E1 -17738.272,E2 -17738.272} C_VEL
LIN {X 0,Y 269.183,Z 752.978,A -85,B 0,C 180,E1 -17740.913,E2 -17740.913} C_VEL
LIN {X 0,Y 269.954,Z 745.349,A -85,B 0,C 180,E1 -17743.169,E2 -17743.169} C_VEL
LIN {X 0,Y 271.055,Z 735.792,A -85,B 0,C 180,E1 -17745.414,E2 -17745.414} C_VEL
LIN {X 0,Y 272.078,Z 726.933,A -85,B 0,C 180,E1 -17747.108,E2 -17747.108} C_VEL
LIN {X 0,Y 273.388,Z 716.407,A -85,B 0,C 180,E1 -17748.745,E2 -17748.745} C_VEL
LIN {X 0,Y 274.073,Z 707.775,A -85,B 0,C 180,E1 -17749.864,E2 -17749.864} C_VEL
LIN {X 0,Y 273.936,Z 695.418,A -85,B 0,C 180,E1 -17751.19,E2 -17751.19} C_VEL
LIN {X 0,Y 273.379,Z 682.816,A -85,B 0,C 180,E1 -17752.257,E2 -17752.257} C_VEL
LIN {X 0,Y 272.776,Z 673.686,A -85,B 0,C 180,E1 -17752.937,E2 -17752.937} C_VEL
LIN {X 0,Y 271.797,Z 660.293,A -85,B 0,C 180,E1 -17753.983,E2 -17753.983} C_VEL
LIN {X 0,Y 270.595,Z 649.732,A -85,B 0,C 180,E1 -17754.626,E2 -17754.626} C_VEL
LIN {X 0,Y 270.229,Z 641.281,A -85,B 0,C 180,E1 -17755.723,E2 -17755.723} C_VEL
LIN {X 0,Y 271.232,Z 632.555,A -85,B 0,C 180,E1 -17759.494,E2 -17759.494} C_VEL
LIN {X 0,Y 272.581,Z 622.971,A -85,B 0,C 180,E1 -17763.656,E2 -17763.656} C_VEL
LIN {X 0,Y 274.168,Z 613.263,A -85,B 0,C 180,E1 -17767.969,E2 -17767.969} C_VEL
LIN {X 0,Y 273.775,Z 609.17,A -85,B 0,C 180,E1 -17769.925,E2 -17769.925} C_VEL
LIN {X 0,Y 272.308,Z 601.556,A -85,B 0,C 180,E1 -17773.725,E2 -17773.725} C_VEL
LIN {X 0,Y 270.89,Z 594.279,A -85,B 0,C 180,E1 -17777.58,E2 -17777.58} C_VEL
LIN {X 0,Y 270.214,Z 590.829,A -85,B 0,C 180,E1 -17779.563,E2 -17779.563} C_VEL
LIN {X 0,Y 270.261,Z 590.825,A -85,B 0,C 180,E1 -17783.722,E2 -17783.722} C_VEL
LIN {X 0,Y 270.21,Z 590.829,A -85,B 0,C 180,E1 -17786.893,E2 -17786.893} C_VEL
LIN {X 0,Y 270.226,Z 590.827,A -85,B 0,C 180,E1 -17790.386,E2 -17790.386} C_VEL
LIN {X 0,Y 270.268,Z 590.818,A -85,B 0,C 180,E1 -17793.764,E2 -17793.764} C_VEL
LIN {X 0,Y 270.242,Z 590.821,A -85,B 0,C 180,E1 -17797.039,E2 -17797.039} C_VEL
LIN {X 0,Y 270.308,Z 590.817,A -85,B 0,C 180,E1 -17800.244,E2 -17800.244} C_VEL
LIN {X 0,Y 270.409,Z 590.802,A -85,B 0,C 180,E1 -17804.935,E2 -17804.935} C_VEL
LIN {X 0,Y 270.447,Z 590.796,A -85,B 0,C 180,E1 -17809.519,E2 -17809.519} C_VEL
LIN {X 0,Y 270.617,Z 590.777,A -85,B 0,C 180,E1 -17812.538,E2 -17812.538} C_VEL
LIN {X 0,Y 270.792,Z 590.755,A -85,B 0,C 180,E1 -17818.512,E2 -17818.512} C_VEL
LIN {X 0,Y 270.792,Z 590.75,A -85,B 0,C 180,E1 -17821.487,E2 -17821.487} C_VEL
LIN {X 0,Y 270.616,Z 590.77,A -85,B 0,C 180,E1 -17827.46,E2 -17827.46} C_VEL
LIN {X 0,Y 270.446,Z 590.799,A -85,B 0,C 180,E1 -17830.48,E2 -17830.48} C_VEL
LIN {X 0,Y 270.4,Z 590.793,A -85,B 0,C 180,E1 -17835.064,E2 -17835.064} C_VEL
LIN {X 0,Y 270.306,Z 590.811,A -85,B 0,C 180,E1 -17839.755,E2 -17839.755} C_VEL
LIN {X 0,Y 270.278,Z 590.814,A -85,B 0,C 180,E1 -17844.585,E2 -17844.585} C_VEL
LIN {X 0,Y 270.275,Z 590.811,A -85,B 0,C 180,E1 -17847.908,E2 -17847.908} C_VEL
LIN {X 0,Y 270.187,Z 590.827,A -85,B 0,C 180,E1 -17851.347,E2 -17851.347} C_VEL
LIN {X 0,Y 270.204,Z 590.826,A -85,B 0,C 180,E1 -17854.904,E2 -17854.904} C_VEL
LIN {X 0,Y 270.2,Z 590.827,A -85,B 0,C 180,E1 -17858.709,E2 -17858.709} C_VEL
LIN {X 0,Y 270.174,Z 590.826,A -85,B 0,C 180,E1 -17863.249,E2 -17863.249} C_VEL
LIN {X 0,Y 270.193,Z 590.825,A -85,B 0,C 180,E1 -17867.445,E2 -17867.445} C_VEL
LIN {X 0,Y 270.208,Z 590.82,A -85,B 0,C 180,E1 -17871.373,E2 -17871.373} C_VEL
LIN {X 0,Y 270.216,Z 590.824,A -85,B 0,C 180,E1 -17875.095,E2 -17875.095} C_VEL
LIN {X 0,Y 270.201,Z 590.825,A -85,B 0,C 180,E1 -17879.129,E2 -17879.129} C_VEL
LIN {X 0,Y 270.263,Z 590.82,A -85,B 0,C 180,E1 -17882.145,E2 -17882.145} C_VEL
LIN {X 0,Y 270.277,Z 590.816,A -85,B 0,C 180,E1 -17885.518,E2 -17885.518} C_VEL
LIN {X 0,Y 270.302,Z 590.815,A -85,B 0,C 180,E1 -17890.243,E2 -17890.243} C_VEL
LIN {X 0,Y 270.403,Z 590.8,A -85,B 0,C 180,E1 -17894.934,E2 -17894.934} C_VEL
LIN {X 0,Y 270.442,Z 590.797,A -85,B 0,C 180,E1 -17899.518,E2 -17899.518} C_VEL
LIN {X 0,Y 270.554,Z 590.785,A -85,B 0,C 180,E1 -17900.541,E2 -17900.541} C_VEL
LIN {X 0,Y 274.589,Z 602.976,A -85,B 0,C 180,E1 -17901.906,E2 -17901.906} C_VEL
LIN {X 0,Y 277.682,Z 614.949,A -85,B 0,C 180,E1 -17903.495,E2 -17903.495} C_VEL
LIN {X 0,Y 278.244,Z 618.119,A -85,B 0,C 180,E1 -17903.963,E2 -17903.963} C_VEL
LIN {X 0,Y 277.098,Z 628.486,A -85,B 0,C 180,E1 -17905.453,E2 -17905.453} C_VEL
LIN {X 0,Y 276,Z 637.637,A -85,B 0,C 180,E1 -17907.079,E2 -17907.079} C_VEL
LIN {X 0,Y 274.71,Z 646.539,A -85,B 0,C 180,E1 -17909.025,E2 -17909.025} C_VEL
LIN {X 0,Y 273.593,Z 654.218,A -85,B 0,C 180,E1 -17911.102,E2 -17911.102} C_VEL
LIN {X 0,Y 272.617,Z 660.836,A -85,B 0,C 180,E1 -17913.324,E2 -17913.324} C_VEL
LIN {X 0,Y 271.667,Z 666.915,A -85,B 0,C 180,E1 -17915.938,E2 -17915.938} C_VEL
LIN {X 0,Y 271.091,Z 670.882,A -85,B 0,C 180,E1 -17918.196,E2 -17918.196} C_VEL
LIN {X 0,Y 270.753,Z 673.82,A -85,B 0,C 180,E1 -17920.467,E2 -17920.467} C_VEL
LIN {X 0,Y 270.677,Z 675.219,A -85,B 0,C 180,E1 -17921.987,E2 -17921.987} C_VEL
LIN {X 0,Y 270.676,Z 676.231,A -85,B 0,C 180,E1 -17923.512,E2 -17923.512} C_VEL
LIN {X 0,Y 271.041,Z 677.021,A -85,B 0,C 180,E1 -17926.385,E2 -17926.385} C_VEL
LIN {X 0,Y 271.346,Z 676.793,A -85,B 0,C 180,E1 -17928.106,E2 -17928.106} C_VEL
LIN {X 0,Y 271.78,Z 676.177,A -85,B 0,C 180,E1 -17929.642,E2 -17929.642} C_VEL
LIN {X 0,Y 272.655,Z 674.477,A -85,B 0,C 180,E1 -17931.886,E2 -17931.886} C_VEL
LIN {X 0,Y 274.27,Z 670.504,A -85,B 0,C 180,E1 -17935.01,E2 -17935.01} C_VEL
LIN {X 0,Y 275.803,Z 666.257,A -85,B 0,C 180,E1 -17937.3,E2 -17937.3} C_VEL
LIN {X 0,Y 277.586,Z 660.732,A -85,B 0,C 180,E1 -17939.583,E2 -17939.583} C_VEL
LIN {X 0,Y 279.716,Z 653.692,A -85,B 0,C 180,E1 -17941.844,E2 -17941.844} C_VEL
LIN {X 0,Y 281.696,Z 646.376,A -85,B 0,C 180,E1 -17943.717,E2 -17943.717} C_VEL
LIN {X 0,Y 283.995,Z 636.68,A -85,B 0,C 180,E1 -17945.71,E2 -17945.71} C_VEL
LIN {X 0,Y 285.094,Z 631.386,A -85,B 0,C 180,E1 -17946.631,E2 -17946.631} C_VEL
LIN {X 0,Y 285.126,Z 629.405,A -85,B 0,C 180,E1 -17946.987,E2 -17946.987} C_VEL
LIN {X 0,Y 283.671,Z 623.905,A -85,B 0,C 180,E1 -17948.131,E2 -17948.131} C_VEL
LIN {X 0,Y 279.235,Z 617.424,A -85,B 0,C 180,E1 -17949.742,E2 -17949.742} C_VEL
LIN {X 0,Y 274.981,Z 612.274,A -85,B 0,C 180,E1 -17951.066,E2 -17951.066} C_VEL
LIN {X 0,Y 273.841,Z 611.413,A -85,B 0,C 180,E1 -17951.351,E2 -17951.351} C_VEL
LIN {X 0,Y 272.779,Z 609.482,A -85,B 0,C 180,E1 -17951.8,E2 -17951.8} C_VEL
LIN {X 0,Y 272.193,Z 617.555,A -85,B 0,C 180,E1 -17955.803,E2 -17955.803} C_VEL
LIN {X 0,Y 271.501,Z 626.917,A -85,B 0,C 180,E1 -17960.394,E2 -17960.394} C_VEL
LIN {X 0,Y 271.174,Z 633.319,A -85,B 0,C 180,E1 -17963.495,E2 -17963.495} C_VEL
LIN {X 0,Y 273.486,Z 646.681,A -85,B 0,C 180,E1 -17964.357,E2 -17964.357} C_VEL
LIN {X 0,Y 275.879,Z 661.209,A -85,B 0,C 180,E1 -17965.627,E2 -17965.627} C_VEL
LIN {X 0,Y 276.42,Z 665.945,A -85,B 0,C 180,E1 -17966.111,E2 -17966.111} C_VEL
LIN {X 0,Y 275.065,Z 678.98,A -85,B 0,C 180,E1 -17967.551,E2 -17967.551} C_VEL
LIN {X 0,Y 273.724,Z 690.122,A -85,B 0,C 180,E1 -17969.103,E2 -17969.103} C_VEL
LIN {X 0,Y 272.478,Z 700.432,A -85,B 0,C 180,E1 -17970.889,E2 -17970.889} C_VEL
LIN {X 0,Y 271.219,Z 710.478,A -85,B 0,C 180,E1 -17973.034,E2 -17973.034} C_VEL
LIN {X 0,Y 270.104,Z 719.288,A -85,B 0,C 180,E1 -17975.399,E2 -17975.399} C_VEL
LIN {X 0,Y 269.358,Z 726.363,A -85,B 0,C 180,E1 -17977.77,E2 -17977.77} C_VEL
LIN {X 0,Y 268.783,Z 732.181,A -85,B 0,C 180,E1 -17980.267,E2 -17980.267} C_VEL
LIN {X 0,Y 268.431,Z 736.153,A -85,B 0,C 180,E1 -17982.478,E2 -17982.478} C_VEL
LIN {X 0,Y 268.241,Z 739.254,A -85,B 0,C 180,E1 -17984.812,E2 -17984.812} C_VEL
LIN {X 0,Y 268.261,Z 740.739,A -85,B 0,C 180,E1 -17986.363,E2 -17986.363} C_VEL
LIN {X 0,Y 268.314,Z 741.797,A -85,B 0,C 180,E1 -17987.905,E2 -17987.905} C_VEL
LIN {X 0,Y 268.458,Z 742.381,A -85,B 0,C 180,E1 -17989.441,E2 -17989.441} C_VEL
LIN {X 0,Y 268.715,Z 742.558,A -85,B 0,C 180,E1 -17990.972,E2 -17990.972} C_VEL
LIN {X 0,Y 269.195,Z 742.253,A -85,B 0,C 180,E1 -17992.772,E2 -17992.772} C_VEL
LIN {X 0,Y 270.047,Z 740.636,A -85,B 0,C 180,E1 -17995.523,E2 -17995.523} C_VEL
LIN {X 0,Y 270.725,Z 739.18,A -85,B 0,C 180,E1 -17997.024,E2 -17997.024} C_VEL
LIN {X 0,Y 272.028,Z 736.19,A -85,B 0,C 180,E1 -17999.26,E2 -17999.26} C_VEL
LIN {X 0,Y 273.628,Z 732.21,A -85,B 0,C 180,E1 -18001.472,E2 -18001.472} C_VEL
LIN {X 0,Y 275.619,Z 727.108,A -85,B 0,C 180,E1 -18003.656,E2 -18003.656} C_VEL
LIN {X 0,Y 277.987,Z 720.741,A -85,B 0,C 180,E1 -18005.805,E2 -18005.805} C_VEL
LIN {X 0,Y 279.987,Z 714.995,A -85,B 0,C 180,E1 -18007.416,E2 -18007.416} C_VEL
LIN {X 0,Y 280.629,Z 711.527,A -85,B 0,C 180,E1 -18008.391,E2 -18008.391} C_VEL
LIN {X 0,Y 280.254,Z 705.863,A -85,B 0,C 180,E1 -18010.06,E2 -18010.06} C_VEL
LIN {X 0,Y 280.029,Z 699.653,A -85,B 0,C 180,E1 -18011.628,E2 -18011.628} C_VEL
LIN {X 0,Y 280.854,Z 695.346,A -85,B 0,C 180,E1 -18012.426,E2 -18012.426} C_VEL
LIN {X 0,Y 284.153,Z 683.474,A -85,B 0,C 180,E1 -18014.138,E2 -18014.138} C_VEL
LIN {X 0,Y 284.443,Z 681.395,A -85,B 0,C 180,E1 -18014.445,E2 -18014.445} C_VEL
LIN {X 0,Y 283.664,Z 672.056,A -85,B 0,C 180,E1 -18016.17,E2 -18016.17} C_VEL
LIN {X 0,Y 281.331,Z 661.047,A -85,B 0,C 180,E1 -18018.331,E2 -18018.331} C_VEL
LIN {X 0,Y 277.448,Z 649.2,A -85,B 0,C 180,E1 -18020.921,E2 -18020.921} C_VEL
LIN {X 0,Y 275.32,Z 644.115,A -85,B 0,C 180,E1 -18022.171,E2 -18022.171} C_VEL
LIN {X 0,Y 274.207,Z 640.864,A -85,B 0,C 180,E1 -18022.969,E2 -18022.969} C_VEL
LIN {X 0,Y 275.492,Z 637.136,A -85,B 0,C 180,E1 -18025.702,E2 -18025.702} C_VEL
LIN {X 0,Y 275.884,Z 635.331,A -85,B 0,C 180,E1 -18027.294,E2 -18027.294} C_VEL
LIN {X 0,Y 276.197,Z 632.759,A -85,B 0,C 180,E1 -18030.104,E2 -18030.104} C_VEL
LIN {X 0,Y 276.394,Z 630.796,A -85,B 0,C 180,E1 -18032.957,E2 -18032.957} C_VEL
LIN {X 0,Y 276.691,Z 629.46,A -85,B 0,C 180,E1 -18035.748,E2 -18035.748} C_VEL
LIN {X 0,Y 277.091,Z 628.872,A -85,B 0,C 180,E1 -18038.165,E2 -18038.165} C_VEL
LIN {X 0,Y 277.315,Z 629.065,A -85,B 0,C 180,E1 -18040.513,E2 -18040.513} C_VEL
LIN {X 0,Y 277.207,Z 630.435,A -85,B 0,C 180,E1 -18043.199,E2 -18043.199} C_VEL
LIN {X 0,Y 277.124,Z 632.218,A -85,B 0,C 180,E1 -18045.243,E2 -18045.243} C_VEL
LIN {X 0,Y 277.239,Z 635.691,A -85,B 0,C 180,E1 -18048.092,E2 -18048.092} C_VEL
LIN {X 0,Y 277.165,Z 638.091,A -85,B 0,C 180,E1 -18049.527,E2 -18049.527} C_VEL
LIN {X 0,Y 276.373,Z 642.662,A -85,B 0,C 180,E1 -18051.466,E2 -18051.466} C_VEL
LIN {X 0,Y 275.279,Z 651.204,A -85,B 0,C 180,E1 -18054.377,E2 -18054.377} C_VEL
LIN {X 0,Y 278.516,Z 663.841,A -85,B 0,C 180,E1 -18056.562,E2 -18056.562} C_VEL
LIN {X 0,Y 280.654,Z 675.76,A -85,B 0,C 180,E1 -18058.366,E2 -18058.366} C_VEL
LIN {X 0,Y 281.531,Z 686.532,A -85,B 0,C 180,E1 -18059.883,E2 -18059.883} C_VEL
LIN {X 0,Y 281.385,Z 694.989,A -85,B 0,C 180,E1 -18061.04,E2 -18061.04} C_VEL
LIN {X 0,Y 279.832,Z 706.045,A -85,B 0,C 180,E1 -18062.503,E2 -18062.503} C_VEL
LIN {X 0,Y 277.351,Z 717.884,A -85,B 0,C 180,E1 -18064.284,E2 -18064.284} C_VEL
LIN {X 0,Y 275.58,Z 724.918,A -85,B 0,C 180,E1 -18065.519,E2 -18065.519} C_VEL
LIN {X 0,Y 272.114,Z 735.461,A -85,B 0,C 180,E1 -18067.609,E2 -18067.609} C_VEL
LIN {X 0,Y 269.202,Z 744.104,A -85,B 0,C 180,E1 -18069.764,E2 -18069.764} C_VEL
LIN {X 0,Y 266.73,Z 751.252,A -85,B 0,C 180,E1 -18071.967,E2 -18071.967} C_VEL
LIN {X 0,Y 264.597,Z 758.018,A -85,B 0,C 180,E1 -18074.598,E2 -18074.598} C_VEL
LIN {X 0,Y 263.048,Z 762.611,A -85,B 0,C 180,E1 -18076.875,E2 -18076.875} C_VEL
LIN {X 0,Y 262.139,Z 766.183,A -85,B 0,C 180,E1 -18079.185,E2 -18079.185} C_VEL
LIN {X 0,Y 261.459,Z 769.496,A -85,B 0,C 180,E1 -18082.278,E2 -18082.278} C_VEL
LIN {X 0,Y 261.295,Z 770.807,A -85,B 0,C 180,E1 -18084.379,E2 -18084.379} C_VEL
LIN {X 0,Y 261.353,Z 771.404,A -85,B 0,C 180,E1 -18086.919,E2 -18086.919} C_VEL
LIN {X 0,Y 261.44,Z 771.227,A -85,B 0,C 180,E1 -18088.461,E2 -18088.461} C_VEL
LIN {X 0,Y 261.769,Z 770.652,A -85,B 0,C 180,E1 -18090.001,E2 -18090.001} C_VEL
LIN {X 0,Y 261.575,Z 769.558,A -85,B 0,C 180,E1 -18091.541,E2 -18091.541} C_VEL
LIN {X 0,Y 261.45,Z 768.033,A -85,B 0,C 180,E1 -18093.083,E2 -18093.083} C_VEL
LIN {X 0,Y 261.532,Z 764.633,A -85,B 0,C 180,E1 -18095.56,E2 -18095.56} C_VEL
LIN {X 0,Y 261.616,Z 760.586,A -85,B 0,C 180,E1 -18097.721,E2 -18097.721} C_VEL
LIN {X 0,Y 261.913,Z 755.034,A -85,B 0,C 180,E1 -18100.046,E2 -18100.046} C_VEL
LIN {X 0,Y 262.501,Z 748.013,A -85,B 0,C 180,E1 -18102.369,E2 -18102.369} C_VEL
LIN {X 0,Y 263.488,Z 739.275,A -85,B 0,C 180,E1 -18104.68,E2 -18104.68} C_VEL
LIN {X 0,Y 264.505,Z 730.341,A -85,B 0,C 180,E1 -18106.598,E2 -18106.598} C_VEL
LIN {X 0,Y 265.973,Z 719.372,A -85,B 0,C 180,E1 -18108.488,E2 -18108.488} C_VEL
LIN {X 0,Y 267.019,Z 709.945,A -85,B 0,C 180,E1 -18109.809,E2 -18109.809} C_VEL
LIN {X 0,Y 267.003,Z 697.879,A -85,B 0,C 180,E1 -18111.22,E2 -18111.22} C_VEL
LIN {X 0,Y 266.488,Z 684.955,A -85,B 0,C 180,E1 -18112.403,E2 -18112.403} C_VEL
LIN {X 0,Y 265.996,Z 676.308,A -85,B 0,C 180,E1 -18113.082,E2 -18113.082} C_VEL
LIN {X 0,Y 265.137,Z 662.757,A -85,B 0,C 180,E1 -18114.259,E2 -18114.259} C_VEL
LIN {X 0,Y 263.586,Z 647.929,A -85,B 0,C 180,E1 -18115.254,E2 -18115.254} C_VEL
LIN {X 0,Y 263.261,Z 640.155,A -85,B 0,C 180,E1 -18116.349,E2 -18116.349} C_VEL
LIN {X 0,Y 264.383,Z 631.214,A -85,B 0,C 180,E1 -18120.337,E2 -18120.337} C_VEL
LIN {X 0,Y 265.957,Z 620.882,A -85,B 0,C 180,E1 -18124.996,E2 -18124.996} C_VEL
LIN {X 0,Y 267.063,Z 614.636,A -85,B 0,C 180,E1 -18127.862,E2 -18127.862} C_VEL
LIN {X 0,Y 266.873,Z 610.866,A -85,B 0,C 180,E1 -18129.665,E2 -18129.665} C_VEL
LIN {X 0,Y 265.447,Z 603.377,A -85,B 0,C 180,E1 -18133.503,E2 -18133.503} C_VEL
LIN {X 0,Y 264.066,Z 596.411,A -85,B 0,C 180,E1 -18137.259,E2 -18137.259} C_VEL
LIN {X 0,Y 263.167,Z 591.708,A -85,B 0,C 180,E1 -18140.013,E2 -18140.013} C_VEL
LIN {X 0,Y 263.196,Z 591.707,A -85,B 0,C 180,E1 -18144.023,E2 -18144.023} C_VEL
LIN {X 0,Y 263.139,Z 591.71,A -85,B 0,C 180,E1 -18147.712,E2 -18147.712} C_VEL
LIN {X 0,Y 263.204,Z 591.699,A -85,B 0,C 180,E1 -18151.784,E2 -18151.784} C_VEL
LIN {X 0,Y 263.232,Z 591.694,A -85,B 0,C 180,E1 -18155.2,E2 -18155.2} C_VEL
LIN {X 0,Y 263.27,Z 591.691,A -85,B 0,C 180,E1 -18159.693,E2 -18159.693} C_VEL
LIN {X 0,Y 263.357,Z 591.683,A -85,B 0,C 180,E1 -18164.522,E2 -18164.522} C_VEL
LIN {X 0,Y 263.379,Z 591.676,A -85,B 0,C 180,E1 -18169.234,E2 -18169.234} C_VEL
LIN {X 0,Y 263.579,Z 591.654,A -85,B 0,C 180,E1 -18172.338,E2 -18172.338} C_VEL
LIN {X 0,Y 263.756,Z 591.632,A -85,B 0,C 180,E1 -18178.473,E2 -18178.473} C_VEL
LIN {X 0,Y 263.756,Z 591.626,A -85,B 0,C 180,E1 -18181.526,E2 -18181.526} C_VEL
LIN {X 0,Y 263.577,Z 591.647,A -85,B 0,C 180,E1 -18187.661,E2 -18187.661} C_VEL
LIN {X 0,Y 263.378,Z 591.677,A -85,B 0,C 180,E1 -18190.765,E2 -18190.765} C_VEL
LIN {X 0,Y 263.349,Z 591.67,A -85,B 0,C 180,E1 -18195.477,E2 -18195.477} C_VEL
LIN {X 0,Y 263.267,Z 591.691,A -85,B 0,C 180,E1 -18200.306,E2 -18200.306} C_VEL
LIN {X 0,Y 263.212,Z 591.69,A -85,B 0,C 180,E1 -18205.29,E2 -18205.29} C_VEL
LIN {X 0,Y 263.183,Z 591.7,A -85,B 0,C 180,E1 -18208.728,E2 -18208.728} C_VEL
LIN {X 0,Y 263.136,Z 591.709,A -85,B 0,C 180,E1 -18212.287,E2 -18212.287} C_VEL
LIN {X 0,Y 263.185,Z 591.701,A -85,B 0,C 180,E1 -18216.762,E2 -18216.762} C_VEL
LIN {X 0,Y 263.127,Z 591.706,A -85,B 0,C 180,E1 -18221.593,E2 -18221.593} C_VEL
LIN {X 0,Y 263.135,Z 591.701,A -85,B 0,C 180,E1 -18226.017,E2 -18226.017} C_VEL
LIN {X 0,Y 263.124,Z 591.708,A -85,B 0,C 180,E1 -18230.13,E2 -18230.13} C_VEL
LIN {X 0,Y 263.189,Z 591.698,A -85,B 0,C 180,E1 -18234.021,E2 -18234.021} C_VEL
LIN {X 0,Y 263.134,Z 591.703,A -85,B 0,C 180,E1 -18237.711,E2 -18237.711} C_VEL
LIN {X 0,Y 263.196,Z 591.698,A -85,B 0,C 180,E1 -18241.784,E2 -18241.784} C_VEL
LIN {X 0,Y 263.226,Z 591.695,A -85,B 0,C 180,E1 -18245.199,E2 -18245.199} C_VEL
LIN {X 0,Y 263.264,Z 591.69,A -85,B 0,C 180,E1 -18249.692,E2 -18249.692} C_VEL
LIN {X 0,Y 263.351,Z 591.677,A -85,B 0,C 180,E1 -18254.521,E2 -18254.521} C_VEL
LIN {X 0,Y 263.374,Z 591.678,A -85,B 0,C 180,E1 -18259.233,E2 -18259.233} C_VEL
LIN {X 0,Y 263.466,Z 591.779,A -85,B 0,C 180,E1 -18260.013,E2 -18260.013} C_VEL
LIN {X 0,Y 267.071,Z 602.255,A -85,B 0,C 180,E1 -18261.21,E2 -18261.21} C_VEL
LIN {X 0,Y 269.475,Z 610.781,A -85,B 0,C 180,E1 -18262.325,E2 -18262.325} C_VEL
LIN {X 0,Y 271.427,Z 618.849,A -85,B 0,C 180,E1 -18263.522,E2 -18263.522} C_VEL
LIN {X 0,Y 270.267,Z 629.861,A -85,B 0,C 180,E1 -18265.151,E2 -18265.151} C_VEL
LIN {X 0,Y 268.978,Z 639.824,A -85,B 0,C 180,E1 -18267.003,E2 -18267.003} C_VEL
LIN {X 0,Y 267.685,Z 648.405,A -85,B 0,C 180,E1 -18268.97,E2 -18268.97} C_VEL
LIN {X 0,Y 266.514,Z 656.044,A -85,B 0,C 180,E1 -18271.132,E2 -18271.132} C_VEL
LIN {X 0,Y 265.695,Z 661.503,A -85,B 0,C 180,E1 -18273.031,E2 -18273.031} C_VEL
LIN {X 0,Y 264.811,Z 666.883,A -85,B 0,C 180,E1 -18275.328,E2 -18275.328} C_VEL
LIN {X 0,Y 264.182,Z 671.095,A -85,B 0,C 180,E1 -18277.642,E2 -18277.642} C_VEL
LIN {X 0,Y 263.818,Z 673.952,A -85,B 0,C 180,E1 -18279.717,E2 -18279.717} C_VEL
LIN {X 0,Y 263.63,Z 676.436,A -85,B 0,C 180,E1 -18282.312,E2 -18282.312} C_VEL
LIN {X 0,Y 263.685,Z 677.391,A -85,B 0,C 180,E1 -18283.878,E2 -18283.878} C_VEL
LIN {X 0,Y 264.04,Z 678.04,A -85,B 0,C 180,E1 -18286.623,E2 -18286.623} C_VEL
LIN {X 0,Y 264.451,Z 677.747,A -85,B 0,C 180,E1 -18288.595,E2 -18288.595} C_VEL
LIN {X 0,Y 264.947,Z 677.061,A -85,B 0,C 180,E1 -18290.17,E2 -18290.17} C_VEL
LIN {X 0,Y 265.804,Z 675.449,A -85,B 0,C 180,E1 -18292.27,E2 -18292.27} C_VEL
LIN {X 0,Y 267.189,Z 672.343,A -85,B 0,C 180,E1 -18294.887,E2 -18294.887} C_VEL
LIN {X 0,Y 268.719,Z 668.384,A -85,B 0,C 180,E1 -18297.225,E2 -18297.225} C_VEL
LIN {X 0,Y 270.88,Z 662.111,A -85,B 0,C 180,E1 -18299.961,E2 -18299.961} C_VEL
LIN {X 0,Y 273.137,Z 655.067,A -85,B 0,C 180,E1 -18302.308,E2 -18302.308} C_VEL
LIN {X 0,Y 275.588,Z 646.412,A -85,B 0,C 180,E1 -18304.545,E2 -18304.545} C_VEL
LIN {X 0,Y 277.875,Z 637.111,A -85,B 0,C 180,E1 -18306.465,E2 -18306.465} C_VEL
LIN {X 0,Y 278.743,Z 632.784,A -85,B 0,C 180,E1 -18307.235,E2 -18307.235} C_VEL
LIN {X 0,Y 278.302,Z 629.683,A -85,B 0,C 180,E1 -18307.884,E2 -18307.884} C_VEL
LIN {X 0,Y 277.729,Z 627.703,A -85,B 0,C 180,E1 -18308.33,E2 -18308.33} C_VEL
LIN {X 0,Y 273.474,Z 621.572,A -85,B 0,C 180,E1 -18309.974,E2 -18309.974} C_VEL
LIN {X 0,Y 269.442,Z 616.958,A -85,B 0,C 180,E1 -18311.293,E2 -18311.293} C_VEL
LIN {X 0,Y 265.821,Z 612.936,A -85,B 0,C 180,E1 -18312.43,E2 -18312.43} C_VEL
LIN {X 0,Y 265.645,Z 612.435,A -85,B 0,C 180,E1 -18312.572,E2 -18312.572} C_VEL
LIN {X 0,Y 265.074,Z 620.13,A -85,B 0,C 180,E1 -18316.422,E2 -18316.422} C_VEL
LIN {X 0,Y 264.494,Z 628.104,A -85,B 0,C 180,E1 -18320.402,E2 -18320.402} C_VEL
LIN {X 0,Y 264.176,Z 633.652,A -85,B 0,C 180,E1 -18323.135,E2 -18323.135} C_VEL
LIN {X 0,Y 266.511,Z 647.325,A -85,B 0,C 180,E1 -18324.04,E2 -18324.04} C_VEL
LIN {X 0,Y 268.788,Z 661.215,A -85,B 0,C 180,E1 -18325.281,E2 -18325.281} C_VEL
LIN {X 0,Y 269.473,Z 665.822,A -85,B 0,C 180,E1 -18325.766,E2 -18325.766} C_VEL
LIN {X 0,Y 268.282,Z 677.746,A -85,B 0,C 180,E1 -18327.094,E2 -18327.094} C_VEL
LIN {X 0,Y 266.736,Z 690.27,A -85,B 0,C 180,E1 -18328.864,E2 -18328.864} C_VEL
LIN {X 0,Y 265.384,Z 701.233,A -85,B 0,C 180,E1 -18330.823,E2 -18330.823} C_VEL
LIN {X 0,Y 264.045,Z 711.503,A -85,B 0,C 180,E1 -18333.098,E2 -18333.098} C_VEL
LIN {X 0,Y 263.053,Z 719.398,A -85,B 0,C 180,E1 -18335.278,E2 -18335.278} C_VEL
LIN {X 0,Y 262.33,Z 726.119,A -85,B 0,C 180,E1 -18337.557,E2 -18337.557} C_VEL
LIN {X 0,Y 261.767,Z 731.869,A -85,B 0,C 180,E1 -18339.994,E2 -18339.994} C_VEL
LIN {X 0,Y 261.29,Z 736.821,A -85,B 0,C 180,E1 -18342.791,E2 -18342.791} C_VEL
LIN {X 0,Y 261.155,Z 740.324,A -85,B 0,C 180,E1 -18345.643,E2 -18345.643} C_VEL
LIN {X 0,Y 261.212,Z 741.849,A -85,B 0,C 180,E1 -18347.571,E2 -18347.571} C_VEL
LIN {X 0,Y 261.325,Z 742.647,A -85,B 0,C 180,E1 -18349.15,E2 -18349.15} C_VEL
LIN {X 0,Y 261.587,Z 743.029,A -85,B 0,C 180,E1 -18350.724,E2 -18350.724} C_VEL
LIN {X 0,Y 262.105,Z 742.854,A -85,B 0,C 180,E1 -18352.78,E2 -18352.78} C_VEL
LIN {X 0,Y 262.942,Z 741.643,A -85,B 0,C 180,E1 -18355.401,E2 -18355.401} C_VEL
LIN {X 0,Y 263.622,Z 740.372,A -85,B 0,C 180,E1 -18356.944,E2 -18356.944} C_VEL
LIN {X 0,Y 264.952,Z 737.693,A -85,B 0,C 180,E1 -18359.241,E2 -18359.241} C_VEL
LIN {X 0,Y 266.598,Z 734.019,A -85,B 0,C 180,E1 -18361.511,E2 -18361.511} C_VEL
LIN {X 0,Y 269.39,Z 727.455,A -85,B 0,C 180,E1 -18364.489,E2 -18364.489} C_VEL
LIN {X 0,Y 271.935,Z 721.112,A -85,B 0,C 180,E1 -18366.679,E2 -18366.679} C_VEL
LIN {X 0,Y 274.876,Z 713.276,A -85,B 0,C 180,E1 -18368.825,E2 -18368.825} C_VEL
LIN {X 0,Y 278.181,Z 703.77,A -85,B 0,C 180,E1 -18370.923,E2 -18370.923} C_VEL
LIN {X 0,Y 280.854,Z 695.346,A -85,B 0,C 180,E1 -18372.426,E2 -18372.426} C_VEL
LIN {X 0,Y 281.488,Z 692.397,A -85,B 0,C 180,E1 -18372.936,E2 -18372.936} C_VEL
LIN {X 0,Y 281.534,Z 688.163,A -85,B 0,C 180,E1 -18373.795,E2 -18373.795} C_VEL
LIN {X 0,Y 280.855,Z 684.268,A -85,B 0,C 180,E1 -18374.711,E2 -18374.711} C_VEL
LIN {X 0,Y 279.428,Z 679.155,A -85,B 0,C 180,E1 -18375.982,E2 -18375.982} C_VEL
LIN {X 0,Y 278.213,Z 673.744,A -85,B 0,C 180,E1 -18377.213,E2 -18377.213} C_VEL
LIN {X 0,Y 276.273,Z 663.875,A -85,B 0,C 180,E1 -18379.312,E2 -18379.312} C_VEL
LIN {X 0,Y 273.677,Z 654.624,A -85,B 0,C 180,E1 -18381.457,E2 -18381.457} C_VEL
LIN {X 0,Y 270.435,Z 645.729,A -85,B 0,C 180,E1 -18383.811,E2 -18383.811} C_VEL
LIN {X 0,Y 268.968,Z 641.672,A -85,B 0,C 180,E1 -18385.023,E2 -18385.023} C_VEL
LIN {X 0,Y 269.845,Z 638.674,A -85,B 0,C 180,E1 -18387.689,E2 -18387.689} C_VEL
LIN {X 0,Y 270.223,Z 636.056,A -85,B 0,C 180,E1 -18390.881,E2 -18390.881} C_VEL
LIN {X 0,Y 270.59,Z 634.383,A -85,B 0,C 180,E1 -18393.788,E2 -18393.788} C_VEL
LIN {X 0,Y 271.059,Z 633.38,A -85,B 0,C 180,E1 -18396.609,E2 -18396.609} C_VEL
LIN {X 0,Y 271.517,Z 633.119,A -85,B 0,C 180,E1 -18399.059,E2 -18399.059} C_VEL
LIN {X 0,Y 271.688,Z 633.738,A -85,B 0,C 180,E1 -18401.398,E2 -18401.398} C_VEL
LIN {X 0,Y 271.603,Z 635.866,A -85,B 0,C 180,E1 -18404.32,E2 -18404.32} C_VEL
LIN {X 0,Y 271.695,Z 639.832,A -85,B 0,C 180,E1 -18407.738,E2 -18407.738} C_VEL
LIN {X 0,Y 271.683,Z 641.838,A -85,B 0,C 180,E1 -18408.956,E2 -18408.956} C_VEL
LIN {X 0,Y 271.039,Z 645.439,A -85,B 0,C 180,E1 -18410.562,E2 -18410.562} C_VEL
LIN {X 0,Y 270.175,Z 650.836,A -85,B 0,C 180,E1 -18412.504,E2 -18412.504} C_VEL
LIN {X 0,Y 272.675,Z 660.625,A -85,B 0,C 180,E1 -18414.474,E2 -18414.474} C_VEL
LIN {X 0,Y 274.702,Z 670.969,A -85,B 0,C 180,E1 -18416.254,E2 -18416.254} C_VEL
LIN {X 0,Y 276.066,Z 682.756,A -85,B 0,C 180,E1 -18418.126,E2 -18418.126} C_VEL
LIN {X 0,Y 276.006,Z 695.721,A -85,B 0,C 180,E1 -18420.042,E2 -18420.042} C_VEL
LIN {X 0,Y 274.323,Z 706.53,A -85,B 0,C 180,E1 -18421.552,E2 -18421.552} C_VEL
LIN {X 0,Y 271.414,Z 718.731,A -85,B 0,C 180,E1 -18423.471,E2 -18423.471} C_VEL
LIN {X 0,Y 269.261,Z 726.547,A -85,B 0,C 180,E1 -18424.905,E2 -18424.905} C_VEL
LIN {X 0,Y 265.64,Z 736.603,A -85,B 0,C 180,E1 -18427.032,E2 -18427.032} C_VEL
LIN {X 0,Y 262.615,Z 744.929,A -85,B 0,C 180,E1 -18429.233,E2 -18429.233} C_VEL
LIN {X 0,Y 260.012,Z 751.819,A -85,B 0,C 180,E1 -18431.484,E2 -18431.484} C_VEL
LIN {X 0,Y 257.752,Z 758.297,A -85,B 0,C 180,E1 -18434.179,E2 -18434.179} C_VEL
LIN {X 0,Y 256.129,Z 762.72,A -85,B 0,C 180,E1 -18436.514,E2 -18436.514} C_VEL
LIN {X 0,Y 255.126,Z 766.138,A -85,B 0,C 180,E1 -18438.884,E2 -18438.884} C_VEL
LIN {X 0,Y 254.39,Z 769.277,A -85,B 0,C 180,E1 -18442.062,E2 -18442.062} C_VEL
LIN {X 0,Y 254.211,Z 770.556,A -85,B 0,C 180,E1 -18444.43,E2 -18444.43} C_VEL
LIN {X 0,Y 254.278,Z 770.931,A -85,B 0,C 180,E1 -18446.833,E2 -18446.833} C_VEL
LIN {X 0,Y 254.355,Z 770.682,A -85,B 0,C 180,E1 -18448.418,E2 -18448.418} C_VEL
LIN {X 0,Y 254.71,Z 770,A -85,B 0,C 180,E1 -18450.001,E2 -18450.001} C_VEL
LIN {X 0,Y 254.493,Z 768.844,A -85,B 0,C 180,E1 -18451.584,E2 -18451.584} C_VEL
LIN {X 0,Y 254.413,Z 766.284,A -85,B 0,C 180,E1 -18453.961,E2 -18453.961} C_VEL
LIN {X 0,Y 254.483,Z 762.624,A -85,B 0,C 180,E1 -18456.344,E2 -18456.344} C_VEL
LIN {X 0,Y 254.637,Z 757.76,A -85,B 0,C 180,E1 -18458.733,E2 -18458.733} C_VEL
LIN {X 0,Y 255.064,Z 751.579,A -85,B 0,C 180,E1 -18461.122,E2 -18461.122} C_VEL
LIN {X 0,Y 255.889,Z 743.808,A -85,B 0,C 180,E1 -18463.502,E2 -18463.502} C_VEL
LIN {X 0,Y 257.021,Z 734.155,A -85,B 0,C 180,E1 -18465.87,E2 -18465.87} C_VEL
LIN {X 0,Y 258.245,Z 724.378,A -85,B 0,C 180,E1 -18467.788,E2 -18467.788} C_VEL
LIN {X 0,Y 259.716,Z 713.159,A -85,B 0,C 180,E1 -18469.566,E2 -18469.566} C_VEL
LIN {X 0,Y 260.014,Z 705.553,A -85,B 0,C 180,E1 -18470.573,E2 -18470.573} C_VEL
LIN {X 0,Y 259.834,Z 693.299,A -85,B 0,C 180,E1 -18471.939,E2 -18471.939} C_VEL
LIN {X 0,Y 259.16,Z 678.067,A -85,B 0,C 180,E1 -18473.298,E2 -18473.298} C_VEL
LIN {X 0,Y 258.41,Z 665.102,A -85,B 0,C 180,E1 -18474.53,E2 -18474.53} C_VEL
LIN {X 0,Y 257.121,Z 651.559,A -85,B 0,C 180,E1 -18475.51,E2 -18475.51} C_VEL
LIN {X 0,Y 256.605,Z 646.953,A -85,B 0,C 180,E1 -18475.815,E2 -18475.815} C_VEL
LIN {X 0,Y 256.308,Z 639.26,A -85,B 0,C 180,E1 -18476.901,E2 -18476.901} C_VEL
LIN {X 0,Y 257.302,Z 631.775,A -85,B 0,C 180,E1 -18480.354,E2 -18480.354} C_VEL
LIN {X 0,Y 258.802,Z 622.271,A -85,B 0,C 180,E1 -18484.771,E2 -18484.771} C_VEL
LIN {X 0,Y 260.118,Z 614.53,A -85,B 0,C 180,E1 -18488.422,E2 -18488.422} C_VEL
LIN {X 0,Y 259.533,Z 610.008,A -85,B 0,C 180,E1 -18490.691,E2 -18490.691} C_VEL
LIN {X 0,Y 257.958,Z 602.182,A -85,B 0,C 180,E1 -18494.897,E2 -18494.897} C_VEL
LIN {X 0,Y 256.595,Z 595.155,A -85,B 0,C 180,E1 -18498.901,E2 -18498.901} C_VEL
LIN {X 0,Y 256.104,Z 592.589,A -85,B 0,C 180,E1 -18500.519,E2 -18500.519} C_VEL
LIN {X 0,Y 256.151,Z 592.584,A -85,B 0,C 180,E1 -18502.87,E2 -18502.87} C_VEL
LIN {X 0,Y 256.091,Z 592.589,A -85,B 0,C 180,E1 -18506.71,E2 -18506.71} C_VEL
LIN {X 0,Y 256.141,Z 592.578,A -85,B 0,C 180,E1 -18511.406,E2 -18511.406} C_VEL
LIN {X 0,Y 256.174,Z 592.574,A -85,B 0,C 180,E1 -18515.699,E2 -18515.699} C_VEL
LIN {X 0,Y 256.175,Z 592.574,A -85,B 0,C 180,E1 -18519.105,E2 -18519.105} C_VEL
LIN {X 0,Y 256.306,Z 592.56,A -85,B 0,C 180,E1 -18524.085,E2 -18524.085} C_VEL
LIN {X 0,Y 256.315,Z 592.557,A -85,B 0,C 180,E1 -18528.934,E2 -18528.934} C_VEL
LIN {X 0,Y 256.546,Z 592.529,A -85,B 0,C 180,E1 -18532.127,E2 -18532.127} C_VEL
LIN {X 0,Y 256.719,Z 592.509,A -85,B 0,C 180,E1 -18538.431,E2 -18538.431} C_VEL
LIN {X 0,Y 256.719,Z 592.503,A -85,B 0,C 180,E1 -18541.568,E2 -18541.568} C_VEL
LIN {X 0,Y 256.545,Z 592.524,A -85,B 0,C 180,E1 -18547.872,E2 -18547.872} C_VEL
LIN {X 0,Y 256.314,Z 592.555,A -85,B 0,C 180,E1 -18551.065,E2 -18551.065} C_VEL
LIN {X 0,Y 256.299,Z 592.549,A -85,B 0,C 180,E1 -18555.914,E2 -18555.914} C_VEL
LIN {X 0,Y 256.171,Z 592.574,A -85,B 0,C 180,E1 -18560.894,E2 -18560.894} C_VEL
LIN {X 0,Y 256.192,Z 592.565,A -85,B 0,C 180,E1 -18565.137,E2 -18565.137} C_VEL
LIN {X 0,Y 256.117,Z 592.578,A -85,B 0,C 180,E1 -18569.598,E2 -18569.598} C_VEL
LIN {X 0,Y 256.07,Z 592.584,A -85,B 0,C 180,E1 -18573.292,E2 -18573.292} C_VEL
LIN {X 0,Y 256.117,Z 592.579,A -85,B 0,C 180,E1 -18577.27,E2 -18577.27} C_VEL
LIN {X 0,Y 256.057,Z 592.587,A -85,B 0,C 180,E1 -18581.202,E2 -18581.202} C_VEL
LIN {X 0,Y 256.067,Z 592.579,A -85,B 0,C 180,E1 -18585.527,E2 -18585.527} C_VEL
LIN {X 0,Y 256.077,Z 592.586,A -85,B 0,C 180,E1 -18588.799,E2 -18588.799} C_VEL
LIN {X 0,Y 256.146,Z 592.575,A -85,B 0,C 180,E1 -18592.869,E2 -18592.869} C_VEL
LIN {X 0,Y 256.086,Z 592.584,A -85,B 0,C 180,E1 -18596.709,E2 -18596.709} C_VEL
LIN {X 0,Y 256.127,Z 592.579,A -85,B 0,C 180,E1 -18601.408,E2 -18601.408} C_VEL
LIN {X 0,Y 256.168,Z 592.574,A -85,B 0,C 180,E1 -18605.698,E2 -18605.698} C_VEL
LIN {X 0,Y 256.167,Z 592.575,A -85,B 0,C 180,E1 -18609.104,E2 -18609.104} C_VEL
LIN {X 0,Y 256.3,Z 592.555,A -85,B 0,C 180,E1 -18614.084,E2 -18614.084} C_VEL
LIN {X 0,Y 256.31,Z 592.556,A -85,B 0,C 180,E1 -18618.933,E2 -18618.933} C_VEL
LIN {X 0,Y 256.342,Z 592.554,A -85,B 0,C 180,E1 -18619.423,E2 -18619.423} C_VEL
LIN {X 0,Y 260.59,Z 604.822,A -85,B 0,C 180,E1 -18620.909,E2 -18620.909} C_VEL
LIN {X 0,Y 263.044,Z 613.691,A -85,B 0,C 180,E1 -18622.136,E2 -18622.136} C_VEL
LIN {X 0,Y 264.639,Z 620.384,A -85,B 0,C 180,E1 -18623.18,E2 -18623.18} C_VEL
LIN {X 0,Y 263.419,Z 631.202,A -85,B 0,C 180,E1 -18624.832,E2 -18624.832} C_VEL
LIN {X 0,Y 262.202,Z 640.216,A -85,B 0,C 180,E1 -18626.541,E2 -18626.541} C_VEL
LIN {X 0,Y 260.93,Z 648.502,A -85,B 0,C 180,E1 -18628.455,E2 -18628.455} C_VEL
LIN {X 0,Y 259.645,Z 656.62,A -85,B 0,C 180,E1 -18630.774,E2 -18630.774} C_VEL
LIN {X 0,Y 258.587,Z 663.177,A -85,B 0,C 180,E1 -18633.114,E2 -18633.114} C_VEL
LIN {X 0,Y 257.723,Z 668.425,A -85,B 0,C 180,E1 -18635.475,E2 -18635.475} C_VEL
LIN {X 0,Y 257.109,Z 672.518,A -85,B 0,C 180,E1 -18637.854,E2 -18637.854} C_VEL
LIN {X 0,Y 256.776,Z 675.087,A -85,B 0,C 180,E1 -18639.831,E2 -18639.831} C_VEL
LIN {X 0,Y 256.614,Z 677.645,A -85,B 0,C 180,E1 -18642.655,E2 -18642.655} C_VEL
LIN {X 0,Y 256.678,Z 678.516,A -85,B 0,C 180,E1 -18644.264,E2 -18644.264} C_VEL
LIN {X 0,Y 257.174,Z 679.028,A -85,B 0,C 180,E1 -18647.492,E2 -18647.492} C_VEL
LIN {X 0,Y 257.569,Z 678.701,A -85,B 0,C 180,E1 -18649.111,E2 -18649.111} C_VEL
LIN {X 0,Y 258.118,Z 677.913,A -85,B 0,C 180,E1 -18650.728,E2 -18650.728} C_VEL
LIN {X 0,Y 258.96,Z 676.429,A -85,B 0,C 180,E1 -18652.672,E2 -18652.672} C_VEL
LIN {X 0,Y 260.574,Z 672.974,A -85,B 0,C 180,E1 -18655.563,E2 -18655.563} C_VEL
LIN {X 0,Y 262.294,Z 668.68,A -85,B 0,C 180,E1 -18658.062,E2 -18658.062} C_VEL
LIN {X 0,Y 264.562,Z 662.481,A -85,B 0,C 180,E1 -18660.753,E2 -18660.753} C_VEL
LIN {X 0,Y 266.936,Z 655.268,A -85,B 0,C 180,E1 -18663.134,E2 -18663.134} C_VEL
LIN {X 0,Y 269.476,Z 646.581,A -85,B 0,C 180,E1 -18665.385,E2 -18665.385} C_VEL
LIN {X 0,Y 271.721,Z 637.841,A -85,B 0,C 180,E1 -18667.197,E2 -18667.197} C_VEL
LIN {X 0,Y 272.38,Z 634.581,A -85,B 0,C 180,E1 -18667.79,E2 -18667.79} C_VEL
LIN {X 0,Y 271.729,Z 631.406,A -85,B 0,C 180,E1 -18668.521,E2 -18668.521} C_VEL
LIN {X 0,Y 267.353,Z 625.243,A -85,B 0,C 180,E1 -18670.331,E2 -18670.331} C_VEL
LIN {X 0,Y 261.07,Z 618.475,A -85,B 0,C 180,E1 -18672.447,E2 -18672.447} C_VEL
LIN {X 0,Y 258.891,Z 616.253,A -85,B 0,C 180,E1 -18673.151,E2 -18673.151} C_VEL
LIN {X 0,Y 258.543,Z 615.355,A -85,B 0,C 180,E1 -18673.353,E2 -18673.353} C_VEL
LIN {X 0,Y 257.913,Z 622.666,A -85,B 0,C 180,E1 -18677.06,E2 -18677.06} C_VEL
LIN {X 0,Y 257.301,Z 632.129,A -85,B 0,C 180,E1 -18681.823,E2 -18681.823} C_VEL
LIN {X 0,Y 257.229,Z 634.174,A -85,B 0,C 180,E1 -18682.767,E2 -18682.767} C_VEL
LIN {X 0,Y 259.489,Z 647.539,A -85,B 0,C 180,E1 -18683.682,E2 -18683.682} C_VEL
LIN {X 0,Y 261.794,Z 661.993,A -85,B 0,C 180,E1 -18685.015,E2 -18685.015} C_VEL
LIN {X 0,Y 262.431,Z 667.346,A -85,B 0,C 180,E1 -18685.594,E2 -18685.594} C_VEL
LIN {X 0,Y 261.054,Z 679.858,A -85,B 0,C 180,E1 -18687.07,E2 -18687.07} C_VEL
LIN {X 0,Y 259.627,Z 691.641,A -85,B 0,C 180,E1 -18688.822,E2 -18688.822} C_VEL
LIN {X 0,Y 258.182,Z 702.677,A -85,B 0,C 180,E1 -18690.885,E2 -18690.885} C_VEL
LIN {X 0,Y 257.086,Z 710.877,A -85,B 0,C 180,E1 -18692.749,E2 -18692.749} C_VEL
LIN {X 0,Y 256.074,Z 718.756,A -85,B 0,C 180,E1 -18694.912,E2 -18694.912} C_VEL
LIN {X 0,Y 255.279,Z 725.86,A -85,B 0,C 180,E1 -18697.33,E2 -18697.33} C_VEL
LIN {X 0,Y 254.72,Z 731.497,A -85,B 0,C 180,E1 -18699.729,E2 -18699.729} C_VEL
LIN {X 0,Y 254.26,Z 736.215,A -85,B 0,C 180,E1 -18702.3,E2 -18702.3} C_VEL
LIN {X 0,Y 254.108,Z 738.568,A -85,B 0,C 180,E1 -18703.945,E2 -18703.945} C_VEL
LIN {X 0,Y 254.059,Z 740.427,A -85,B 0,C 180,E1 -18705.584,E2 -18705.584} C_VEL
LIN {X 0,Y 254.1,Z 741.862,A -85,B 0,C 180,E1 -18707.217,E2 -18707.217} C_VEL
LIN {X 0,Y 254.195,Z 742.833,A -85,B 0,C 180,E1 -18708.841,E2 -18708.841} C_VEL
LIN {X 0,Y 254.445,Z 743.373,A -85,B 0,C 180,E1 -18710.461,E2 -18710.461} C_VEL
LIN {X 0,Y 255.028,Z 743.436,A -85,B 0,C 180,E1 -18712.769,E2 -18712.769} C_VEL
LIN {X 0,Y 255.817,Z 742.56,A -85,B 0,C 180,E1 -18715.273,E2 -18715.273} C_VEL
LIN {X 0,Y 257.356,Z 740.011,A -85,B 0,C 180,E1 -18718.436,E2 -18718.436} C_VEL
LIN {X 0,Y 259.543,Z 735.751,A -85,B 0,C 180,E1 -18721.552,E2 -18721.552} C_VEL
LIN {X 0,Y 261.645,Z 731.379,A -85,B 0,C 180,E1 -18723.851,E2 -18723.851} C_VEL
LIN {X 0,Y 264.561,Z 724.841,A -85,B 0,C 180,E1 -18726.483,E2 -18726.483} C_VEL
LIN {X 0,Y 268.01,Z 716.516,A -85,B 0,C 180,E1 -18729.053,E2 -18729.053} C_VEL
LIN {X 0,Y 271.477,Z 707.605,A -85,B 0,C 180,E1 -18731.196,E2 -18731.196} C_VEL
LIN {X 0,Y 275.276,Z 696.596,A -85,B 0,C 180,E1 -18733.285,E2 -18733.285} C_VEL
LIN {X 0,Y 278.511,Z 685.94,A -85,B 0,C 180,E1 -18734.899,E2 -18734.899} C_VEL
LIN {X 0,Y 278.932,Z 684.15,A -85,B 0,C 180,E1 -18735.158,E2 -18735.158} C_VEL
LIN {X 0,Y 278.297,Z 674.32,A -85,B 0,C 180,E1 -18737.095,E2 -18737.095} C_VEL
LIN {X 0,Y 278.213,Z 673.744,A -85,B 0,C 180,E1 -18737.213,E2 -18737.213} C_VEL
LIN {X 0,Y 277.112,Z 670.033,A -85,B 0,C 180,E1 -18738.13,E2 -18738.13} C_VEL
LIN {X 0,Y 275.332,Z 667.045,A -85,B 0,C 180,E1 -18739.129,E2 -18739.129} C_VEL
LIN {X 0,Y 270.008,Z 659.987,A -85,B 0,C 180,E1 -18741.943,E2 -18741.943} C_VEL
LIN {X 0,Y 269.082,Z 657.813,A -85,B 0,C 180,E1 -18742.632,E2 -18742.632} C_VEL
LIN {X 0,Y 266.927,Z 650.89,A -85,B 0,C 180,E1 -18744.583,E2 -18744.583} C_VEL
LIN {X 0,Y 265.501,Z 646.924,A -85,B 0,C 180,E1 -18745.846,E2 -18745.846} C_VEL
LIN {X 0,Y 263.708,Z 642.569,A -85,B 0,C 180,E1 -18747.593,E2 -18747.593} C_VEL
LIN {X 0,Y 264.205,Z 640.352,A -85,B 0,C 180,E1 -18750.359,E2 -18750.359} C_VEL
LIN {X 0,Y 264.785,Z 638.418,A -85,B 0,C 180,E1 -18753.876,E2 -18753.876} C_VEL
LIN {X 0,Y 265.5,Z 637.458,A -85,B 0,C 180,E1 -18757.506,E2 -18757.506} C_VEL
LIN {X 0,Y 265.985,Z 637.615,A -85,B 0,C 180,E1 -18759.984,E2 -18759.984} C_VEL
LIN {X 0,Y 266.075,Z 638.74,A -85,B 0,C 180,E1 -18762.307,E2 -18762.307} C_VEL
LIN {X 0,Y 266.025,Z 641.624,A -85,B 0,C 180,E1 -18765.505,E2 -18765.505} C_VEL
LIN {X 0,Y 266.172,Z 644.421,A -85,B 0,C 180,E1 -18767.674,E2 -18767.674} C_VEL
LIN {X 0,Y 266.122,Z 646.137,A -85,B 0,C 180,E1 -18768.685,E2 -18768.685} C_VEL
LIN {X 0,Y 265.436,Z 650.032,A -85,B 0,C 180,E1 -18770.363,E2 -18770.363} C_VEL
LIN {X 0,Y 268.254,Z 662.507,A -85,B 0,C 180,E1 -18773.132,E2 -18773.132} C_VEL
LIN {X 0,Y 269.956,Z 672.684,A -85,B 0,C 180,E1 -18775.06,E2 -18775.06} C_VEL
LIN {X 0,Y 270.924,Z 683.964,A -85,B 0,C 180,E1 -18776.994,E2 -18776.994} C_VEL
LIN {X 0,Y 270.789,Z 694.972,A -85,B 0,C 180,E1 -18778.732,E2 -18778.732} C_VEL
LIN {X 0,Y 269.839,Z 702.619,A -85,B 0,C 180,E1 -18779.899,E2 -18779.899} C_VEL
LIN {X 0,Y 266.752,Z 715.631,A -85,B 0,C 180,E1 -18781.906,E2 -18781.906} C_VEL
LIN {X 0,Y 263.645,Z 726.318,A -85,B 0,C 180,E1 -18783.908,E2 -18783.908} C_VEL
LIN {X 0,Y 259.815,Z 736.308,A -85,B 0,C 180,E1 -18786.064,E2 -18786.064} C_VEL
LIN {X 0,Y 256.527,Z 744.541,A -85,B 0,C 180,E1 -18788.295,E2 -18788.295} C_VEL
LIN {X 0,Y 253.299,Z 752.363,A -85,B 0,C 180,E1 -18790.975,E2 -18790.975} C_VEL
LIN {X 0,Y 250.928,Z 758.649,A -85,B 0,C 180,E1 -18793.737,E2 -18793.737} C_VEL
LIN {X 0,Y 249.228,Z 762.86,A -85,B 0,C 180,E1 -18796.133,E2 -18796.133} C_VEL
LIN {X 0,Y 248.132,Z 766.103,A -85,B 0,C 180,E1 -18798.566,E2 -18798.566} C_VEL
LIN {X 0,Y 247.644,Z 767.775,A -85,B 0,C 180,E1 -18800.198,E2 -18800.198} C_VEL
LIN {X 0,Y 247.172,Z 769.885,A -85,B 0,C 180,E1 -18803.471,E2 -18803.471} C_VEL
LIN {X 0,Y 247.12,Z 770.366,A -85,B 0,C 180,E1 -18805.107,E2 -18805.107} C_VEL
LIN {X 0,Y 247.203,Z 770.45,A -85,B 0,C 180,E1 -18806.742,E2 -18806.742} C_VEL
LIN {X 0,Y 247.65,Z 769.328,A -85,B 0,C 180,E1 -18810.001,E2 -18810.001} C_VEL
LIN {X 0,Y 247.413,Z 768.102,A -85,B 0,C 180,E1 -18811.629,E2 -18811.629} C_VEL
LIN {X 0,Y 247.358,Z 765.406,A -85,B 0,C 180,E1 -18814.075,E2 -18814.075} C_VEL
LIN {X 0,Y 247.427,Z 761.618,A -85,B 0,C 180,E1 -18816.525,E2 -18816.525} C_VEL
LIN {X 0,Y 247.594,Z 756.617,A -85,B 0,C 180,E1 -18818.983,E2 -18818.983} C_VEL
LIN {X 0,Y 248.066,Z 750.241,A -85,B 0,C 180,E1 -18821.44,E2 -18821.44} C_VEL
LIN {X 0,Y 248.93,Z 742.267,A -85,B 0,C 180,E1 -18823.887,E2 -18823.887} C_VEL
LIN {X 0,Y 249.911,Z 734.145,A -85,B 0,C 180,E1 -18825.915,E2 -18825.915} C_VEL
LIN {X 0,Y 251.2,Z 724.059,A -85,B 0,C 180,E1 -18827.964,E2 -18827.964} C_VEL
LIN {X 0,Y 252.796,Z 712.043,A -85,B 0,C 180,E1 -18829.913,E2 -18829.913} C_VEL
LIN {X 0,Y 252.961,Z 700.745,A -85,B 0,C 180,E1 -18831.388,E2 -18831.388} C_VEL
LIN {X 0,Y 252.634,Z 688.223,A -85,B 0,C 180,E1 -18832.706,E2 -18832.706} C_VEL
LIN {X 0,Y 252.282,Z 680.733,A -85,B 0,C 180,E1 -18833.39,E2 -18833.39} C_VEL
LIN {X 0,Y 251.75,Z 667.812,A -85,B 0,C 180,E1 -18834.757,E2 -18834.757} C_VEL
LIN {X 0,Y 250.631,Z 654.627,A -85,B 0,C 180,E1 -18835.829,E2 -18835.829} C_VEL
LIN {X 0,Y 249.616,Z 645.791,A -85,B 0,C 180,E1 -18836.412,E2 -18836.412} C_VEL
LIN {X 0,Y 249.387,Z 638.165,A -85,B 0,C 180,E1 -18837.597,E2 -18837.597} C_VEL
LIN {X 0,Y 250.777,Z 628.544,A -85,B 0,C 180,E1 -18842.174,E2 -18842.174} C_VEL
LIN {X 0,Y 252.481,Z 618.875,A -85,B 0,C 180,E1 -18846.818,E2 -18846.818} C_VEL
LIN {X 0,Y 253.041,Z 614.57,A -85,B 0,C 180,E1 -18848.951,E2 -18848.951} C_VEL
LIN {X 0,Y 252.091,Z 608.825,A -85,B 0,C 180,E1 -18851.999,E2 -18851.999} C_VEL
LIN {X 0,Y 250.387,Z 600.179,A -85,B 0,C 180,E1 -18856.87,E2 -18856.87} C_VEL
LIN {X 0,Y 249.084,Z 593.464,A -85,B 0,C 180,E1 -18860.982,E2 -18860.982} C_VEL
LIN {X 0,Y 249.081,Z 593.464,A -85,B 0,C 180,E1 -18864.913,E2 -18864.913} C_VEL
LIN {X 0,Y 249.057,Z 593.462,A -85,B 0,C 180,E1 -18869.473,E2 -18869.473} C_VEL
LIN {X 0,Y 249.079,Z 593.457,A -85,B 0,C 180,E1 -18873.162,E2 -18873.162} C_VEL
LIN {X 0,Y 249.087,Z 593.458,A -85,B 0,C 180,E1 -18876.733,E2 -18876.733} C_VEL
LIN {X 0,Y 249.118,Z 593.457,A -85,B 0,C 180,E1 -18880.211,E2 -18880.211} C_VEL
LIN {X 0,Y 249.248,Z 593.438,A -85,B 0,C 180,E1 -18883.622,E2 -18883.622} C_VEL
LIN {X 0,Y 249.259,Z 593.438,A -85,B 0,C 180,E1 -18888.616,E2 -18888.616} C_VEL
LIN {X 0,Y 249.49,Z 593.407,A -85,B 0,C 180,E1 -18891.902,E2 -18891.902} C_VEL
LIN {X 0,Y 249.44,Z 593.412,A -85,B 0,C 180,E1 -18896.769,E2 -18896.769} C_VEL
LIN {X 0,Y 249.734,Z 593.377,A -85,B 0,C 180,E1 -18899.999,E2 -18899.999} C_VEL
LIN {X 0,Y 249.439,Z 593.404,A -85,B 0,C 180,E1 -18903.23,E2 -18903.23} C_VEL
LIN {X 0,Y 249.486,Z 593.404,A -85,B 0,C 180,E1 -18908.096,E2 -18908.096} C_VEL
LIN {X 0,Y 249.257,Z 593.434,A -85,B 0,C 180,E1 -18911.383,E2 -18911.383} C_VEL
LIN {X 0,Y 249.222,Z 593.431,A -85,B 0,C 180,E1 -18916.502,E2 -18916.502} C_VEL
LIN {X 0,Y 249.091,Z 593.455,A -85,B 0,C 180,E1 -18921.517,E2 -18921.517} C_VEL
LIN {X 0,Y 249.134,Z 593.443,A -85,B 0,C 180,E1 -18925.481,E2 -18925.481} C_VEL
LIN {X 0,Y 249.087,Z 593.454,A -85,B 0,C 180,E1 -18928.992,E2 -18928.992} C_VEL
LIN {X 0,Y 249.034,Z 593.466,A -85,B 0,C 180,E1 -18932.425,E2 -18932.425} C_VEL
LIN {X 0,Y 249.051,Z 593.463,A -85,B 0,C 180,E1 -18936.341,E2 -18936.341} C_VEL
LIN {X 0,Y 249.008,Z 593.469,A -85,B 0,C 180,E1 -18940.477,E2 -18940.477} C_VEL
LIN {X 0,Y 249.011,Z 593.459,A -85,B 0,C 180,E1 -18944.876,E2 -18944.876} C_VEL
LIN {X 0,Y 249.038,Z 593.46,A -85,B 0,C 180,E1 -18947.366,E2 -18947.366} C_VEL
LIN {X 0,Y 249.041,Z 593.456,A -85,B 0,C 180,E1 -18951.621,E2 -18951.621} C_VEL
LIN {X 0,Y 249.063,Z 593.459,A -85,B 0,C 180,E1 -18955.641,E2 -18955.641} C_VEL
LIN {X 0,Y 249.048,Z 593.459,A -85,B 0,C 180,E1 -18959.471,E2 -18959.471} C_VEL
LIN {X 0,Y 249.072,Z 593.456,A -85,B 0,C 180,E1 -18963.161,E2 -18963.161} C_VEL
LIN {X 0,Y 249.08,Z 593.457,A -85,B 0,C 180,E1 -18966.731,E2 -18966.731} C_VEL
LIN {X 0,Y 249.111,Z 593.455,A -85,B 0,C 180,E1 -18970.21,E2 -18970.21} C_VEL
LIN {X 0,Y 249.242,Z 593.435,A -85,B 0,C 180,E1 -18973.62,E2 -18973.62} C_VEL
LIN {X 0,Y 249.274,Z 593.431,A -85,B 0,C 180,E1 -18978.784,E2 -18978.784} C_VEL
LIN {X 0,Y 253.761,Z 606.21,A -85,B 0,C 180,E1 -18980.433,E2 -18980.433} C_VEL
LIN {X 0,Y 256.257,Z 615.116,A -85,B 0,C 180,E1 -18981.72,E2 -18981.72} C_VEL
LIN {X 0,Y 257.841,Z 621.985,A -85,B 0,C 180,E1 -18982.828,E2 -18982.828} C_VEL
LIN {X 0,Y 256.584,Z 632.527,A -85,B 0,C 180,E1 -18984.497,E2 -18984.497} C_VEL
LIN {X 0,Y 255.161,Z 642.37,A -85,B 0,C 180,E1 -18986.446,E2 -18986.446} C_VEL
LIN {X 0,Y 253.86,Z 650.47,A -85,B 0,C 180,E1 -18988.412,E2 -18988.412} C_VEL
LIN {X 0,Y 252.574,Z 658.424,A -85,B 0,C 180,E1 -18990.796,E2 -18990.796} C_VEL
LIN {X 0,Y 251.49,Z 664.823,A -85,B 0,C 180,E1 -18993.202,E2 -18993.202} C_VEL
LIN {X 0,Y 250.613,Z 669.925,A -85,B 0,C 180,E1 -18995.631,E2 -18995.631} C_VEL
LIN {X 0,Y 250.02,Z 673.898,A -85,B 0,C 180,E1 -18998.078,E2 -18998.078} C_VEL
LIN {X 0,Y 249.729,Z 676.213,A -85,B 0,C 180,E1 -18999.945,E2 -18999.945} C_VEL
LIN {X 0,Y 249.598,Z 678.836,A -85,B 0,C 180,E1 -19003.016,E2 -19003.016} C_VEL
LIN {X 0,Y 249.934,Z 680.021,A -85,B 0,C 180,E1 -19006.33,E2 -19006.33} C_VEL
LIN {X 0,Y 250.278,Z 680.035,A -85,B 0,C 180,E1 -19007.991,E2 -19007.991} C_VEL
LIN {X 0,Y 250.722,Z 679.611,A -85,B 0,C 180,E1 -19009.654,E2 -19009.654} C_VEL
LIN {X 0,Y 251.314,Z 678.765,A -85,B 0,C 180,E1 -19011.316,E2 -19011.316} C_VEL
LIN {X 0,Y 252.13,Z 677.408,A -85,B 0,C 180,E1 -19013.096,E2 -19013.096} C_VEL
LIN {X 0,Y 253.472,Z 674.766,A -85,B 0,C 180,E1 -19015.451,E2 -19015.451} C_VEL
LIN {X 0,Y 255.44,Z 670.215,A -85,B 0,C 180,E1 -19018.308,E2 -19018.308} C_VEL
LIN {X 0,Y 257.505,Z 664.872,A -85,B 0,C 180,E1 -19020.778,E2 -19020.778} C_VEL
LIN {X 0,Y 259.654,Z 658.857,A -85,B 0,C 180,E1 -19022.959,E2 -19022.959} C_VEL
LIN {X 0,Y 262.137,Z 651.126,A -85,B 0,C 180,E1 -19025.197,E2 -19025.197} C_VEL
LIN {X 0,Y 264.579,Z 642.614,A -85,B 0,C 180,E1 -19027.167,E2 -19027.167} C_VEL
LIN {X 0,Y 265.911,Z 637.223,A -85,B 0,C 180,E1 -19028.216,E2 -19028.216} C_VEL
LIN {X 0,Y 265.858,Z 635.753,A -85,B 0,C 180,E1 -19028.543,E2 -19028.543} C_VEL
LIN {X 0,Y 263.186,Z 631.456,A -85,B 0,C 180,E1 -19029.856,E2 -19029.856} C_VEL
LIN {X 0,Y 258.236,Z 625.712,A -85,B 0,C 180,E1 -19031.754,E2 -19031.754} C_VEL
LIN {X 0,Y 251.711,Z 619.244,A -85,B 0,C 180,E1 -19034.014,E2 -19034.014} C_VEL
LIN {X 0,Y 251.406,Z 618.422,A -85,B 0,C 180,E1 -19034.22,E2 -19034.22} C_VEL
LIN {X 0,Y 250.684,Z 626.845,A -85,B 0,C 180,E1 -19038.555,E2 -19038.555} C_VEL
LIN {X 0,Y 250.231,Z 634.434,A -85,B 0,C 180,E1 -19042.371,E2 -19042.371} C_VEL
LIN {X 0,Y 252.49,Z 647.908,A -85,B 0,C 180,E1 -19043.317,E2 -19043.317} C_VEL
LIN {X 0,Y 254.735,Z 662.381,A -85,B 0,C 180,E1 -19044.693,E2 -19044.693} C_VEL
LIN {X 0,Y 255.472,Z 667.118,A -85,B 0,C 180,E1 -19045.23,E2 -19045.23} C_VEL
LIN {X 0,Y 254.202,Z 679.192,A -85,B 0,C 180,E1 -19046.669,E2 -19046.669} C_VEL
LIN {X 0,Y 252.771,Z 690.445,A -85,B 0,C 180,E1 -19048.346,E2 -19048.346} C_VEL
LIN {X 0,Y 251.385,Z 701.141,A -85,B 0,C 180,E1 -19050.332,E2 -19050.332} C_VEL
LIN {X 0,Y 250.152,Z 710.152,A -85,B 0,C 180,E1 -19052.383,E2 -19052.383} C_VEL
LIN {X 0,Y 248.972,Z 719.322,A -85,B 0,C 180,E1 -19054.95,E2 -19054.95} C_VEL
LIN {X 0,Y 248.137,Z 726.6,A -85,B 0,C 180,E1 -19057.521,E2 -19057.521} C_VEL
LIN {X 0,Y 247.556,Z 732.388,A -85,B 0,C 180,E1 -19060.083,E2 -19060.083} C_VEL
LIN {X 0,Y 247.133,Z 736.857,A -85,B 0,C 180,E1 -19062.627,E2 -19062.627} C_VEL
LIN {X 0,Y 246.962,Z 740.369,A -85,B 0,C 180,E1 -19065.36,E2 -19065.36} C_VEL
LIN {X 0,Y 247.065,Z 742.913,A -85,B 0,C 180,E1 -19068.515,E2 -19068.515} C_VEL
LIN {X 0,Y 247.296,Z 743.677,A -85,B 0,C 180,E1 -19070.183,E2 -19070.183} C_VEL
LIN {X 0,Y 247.943,Z 744.001,A -85,B 0,C 180,E1 -19072.77,E2 -19072.77} C_VEL
LIN {X 0,Y 248.68,Z 743.414,A -85,B 0,C 180,E1 -19075.137,E2 -19075.137} C_VEL
LIN {X 0,Y 249.366,Z 742.544,A -85,B 0,C 180,E1 -19076.769,E2 -19076.769} C_VEL
LIN {X 0,Y 251.304,Z 739.545,A -85,B 0,C 180,E1 -19080.001,E2 -19080.001} C_VEL
LIN {X 0,Y 253.238,Z 736.047,A -85,B 0,C 180,E1 -19082.485,E2 -19082.485} C_VEL
LIN {X 0,Y 255.421,Z 731.82,A -85,B 0,C 180,E1 -19084.736,E2 -19084.736} C_VEL
LIN {X 0,Y 258.63,Z 725.327,A -85,B 0,C 180,E1 -19087.417,E2 -19087.417} C_VEL
LIN {X 0,Y 261.758,Z 718.315,A -85,B 0,C 180,E1 -19089.661,E2 -19089.661} C_VEL
LIN {X 0,Y 265.377,Z 709.741,A -85,B 0,C 180,E1 -19091.844,E2 -19091.844} C_VEL
LIN {X 0,Y 268.671,Z 701.175,A -85,B 0,C 180,E1 -19093.617,E2 -19093.617} C_VEL
LIN {X 0,Y 271.99,Z 691.367,A -85,B 0,C 180,E1 -19095.265,E2 -19095.265} C_VEL
LIN {X 0,Y 273.432,Z 686.654,A -85,B 0,C 180,E1 -19095.947,E2 -19095.947} C_VEL
LIN {X 0,Y 273.16,Z 677.714,A -85,B 0,C 180,E1 -19097.838,E2 -19097.838} C_VEL
LIN {X 0,Y 271.655,Z 667.96,A -85,B 0,C 180,E1 -19100.057,E2 -19100.057} C_VEL
LIN {X 0,Y 269.585,Z 659.342,A -85,B 0,C 180,E1 -19102.193,E2 -19102.193} C_VEL
LIN {X 0,Y 269.082,Z 657.813,A -85,B 0,C 180,E1 -19102.632,E2 -19102.632} C_VEL
LIN {X 0,Y 267.66,Z 654.855,A -85,B 0,C 180,E1 -19103.683,E2 -19103.683} C_VEL
LIN {X 0,Y 265.853,Z 652.728,A -85,B 0,C 180,E1 -19104.811,E2 -19104.811} C_VEL
LIN {X 0,Y 260.084,Z 647.58,A -85,B 0,C 180,E1 -19108.857,E2 -19108.857} C_VEL
LIN {X 0,Y 258.42,Z 643.899,A -85,B 0,C 180,E1 -19111.114,E2 -19111.114} C_VEL
LIN {X 0,Y 259.139,Z 642.245,A -85,B 0,C 180,E1 -19114.718,E2 -19114.718} C_VEL
LIN {X 0,Y 260.008,Z 641.758,A -85,B 0,C 180,E1 -19118.44,E2 -19118.44} C_VEL
LIN {X 0,Y 260.462,Z 642.349,A -85,B 0,C 180,E1 -19120.932,E2 -19120.932} C_VEL
LIN {X 0,Y 260.499,Z 643.921,A -85,B 0,C 180,E1 -19123.247,E2 -19123.247} C_VEL
LIN {X 0,Y 260.519,Z 646.188,A -85,B 0,C 180,E1 -19125.463,E2 -19125.463} C_VEL
LIN {X 0,Y 260.717,Z 649.276,A -85,B 0,C 180,E1 -19127.683,E2 -19127.683} C_VEL
LIN {X 0,Y 262.341,Z 655.482,A -85,B 0,C 180,E1 -19129.615,E2 -19129.615} C_VEL
LIN {X 0,Y 264.563,Z 667.977,A -85,B 0,C 180,E1 -19132.498,E2 -19132.498} C_VEL
LIN {X 0,Y 265.647,Z 677.652,A -85,B 0,C 180,E1 -19134.408,E2 -19134.408} C_VEL
LIN {X 0,Y 266.06,Z 689.591,A -85,B 0,C 180,E1 -19136.558,E2 -19136.558} C_VEL
LIN {X 0,Y 265.176,Z 700.653,A -85,B 0,C 180,E1 -19138.407,E2 -19138.407} C_VEL
LIN {X 0,Y 262.646,Z 711.48,A -85,B 0,C 180,E1 -19140.109,E2 -19140.109} C_VEL
LIN {X 0,Y 258.69,Z 724.532,A -85,B 0,C 180,E1 -19142.495,E2 -19142.495} C_VEL
LIN {X 0,Y 254.768,Z 734.561,A -85,B 0,C 180,E1 -19144.688,E2 -19144.688} C_VEL
LIN {X 0,Y 251.083,Z 742.951,A -85,B 0,C 180,E1 -19146.931,E2 -19146.931} C_VEL
LIN {X 0,Y 247.861,Z 750.207,A -85,B 0,C 180,E1 -19149.343,E2 -19149.343} C_VEL
LIN {X 0,Y 244.808,Z 757.362,A -85,B 0,C 180,E1 -19152.458,E2 -19152.458} C_VEL
LIN {X 0,Y 242.876,Z 761.729,A -85,B 0,C 180,E1 -19154.906,E2 -19154.906} C_VEL
LIN {X 0,Y 241.819,Z 764.116,A -85,B 0,C 180,E1 -19156.557,E2 -19156.557} C_VEL
LIN {X 0,Y 240.628,Z 767.596,A -85,B 0,C 180,E1 -19159.909,E2 -19159.909} C_VEL
LIN {X 0,Y 240.086,Z 769.555,A -85,B 0,C 180,E1 -19163.277,E2 -19163.277} C_VEL
LIN {X 0,Y 240.059,Z 769.94,A -85,B 0,C 180,E1 -19164.963,E2 -19164.963} C_VEL
LIN {X 0,Y 240.13,Z 769.901,A -85,B 0,C 180,E1 -19166.646,E2 -19166.646} C_VEL
LIN {X 0,Y 240.591,Z 768.658,A -85,B 0,C 180,E1 -19170.002,E2 -19170.002} C_VEL
LIN {X 0,Y 240.337,Z 767.331,A -85,B 0,C 180,E1 -19171.677,E2 -19171.677} C_VEL
LIN {X 0,Y 240.305,Z 764.496,A -85,B 0,C 180,E1 -19174.194,E2 -19174.194} C_VEL
LIN {X 0,Y 240.384,Z 760.537,A -85,B 0,C 180,E1 -19176.717,E2 -19176.717} C_VEL
LIN {X 0,Y 240.645,Z 754.344,A -85,B 0,C 180,E1 -19179.669,E2 -19179.669} C_VEL
LIN {X 0,Y 241.19,Z 747.547,A -85,B 0,C 180,E1 -19182.197,E2 -19182.197} C_VEL
LIN {X 0,Y 242.18,Z 739.03,A -85,B 0,C 180,E1 -19184.711,E2 -19184.711} C_VEL
LIN {X 0,Y 243.247,Z 730.353,A -85,B 0,C 180,E1 -19186.795,E2 -19186.795} C_VEL
LIN {X 0,Y 244.712,Z 719.807,A -85,B 0,C 180,E1 -19188.852,E2 -19188.852} C_VEL
LIN {X 0,Y 245.891,Z 710.863,A -85,B 0,C 180,E1 -19190.278,E2 -19190.278} C_VEL
LIN {X 0,Y 245.94,Z 699.345,A -85,B 0,C 180,E1 -19191.809,E2 -19191.809} C_VEL
LIN {X 0,Y 245.569,Z 686.721,A -85,B 0,C 180,E1 -19193.156,E2 -19193.156} C_VEL
LIN {X 0,Y 245.367,Z 680.226,A -85,B 0,C 180,E1 -19193.866,E2 -19193.866} C_VEL
LIN {X 0,Y 244.83,Z 667.407,A -85,B 0,C 180,E1 -19195.279,E2 -19195.279} C_VEL
LIN {X 0,Y 243.752,Z 654.136,A -85,B 0,C 180,E1 -19196.412,E2 -19196.412} C_VEL
LIN {X 0,Y 242.622,Z 644.149,A -85,B 0,C 180,E1 -19197.108,E2 -19197.108} C_VEL
LIN {X 0,Y 242.482,Z 637.25,A -85,B 0,C 180,E1 -19198.217,E2 -19198.217} C_VEL
LIN {X 0,Y 244.017,Z 627.165,A -85,B 0,C 180,E1 -19203.178,E2 -19203.178} C_VEL
LIN {X 0,Y 245.867,Z 617.662,A -85,B 0,C 180,E1 -19207.922,E2 -19207.922} C_VEL
LIN {X 0,Y 245.929,Z 614.638,A -85,B 0,C 180,E1 -19209.502,E2 -19209.502} C_VEL
LIN {X 0,Y 244.804,Z 608.587,A -85,B 0,C 180,E1 -19212.817,E2 -19212.817} C_VEL
LIN {X 0,Y 243.309,Z 601.036,A -85,B 0,C 180,E1 -19217.249,E2 -19217.249} C_VEL
LIN {X 0,Y 242.02,Z 594.344,A -85,B 0,C 180,E1 -19221.521,E2 -19221.521} C_VEL
LIN {X 0,Y 242.043,Z 594.343,A -85,B 0,C 180,E1 -19224.498,E2 -19224.498} C_VEL
LIN {X 0,Y 241.982,Z 594.346,A -85,B 0,C 180,E1 -19228.48,E2 -19228.48} C_VEL
LIN {X 0,Y 242.013,Z 594.34,A -85,B 0,C 180,E1 -19232.313,E2 -19232.313} C_VEL
LIN {X 0,Y 242.064,Z 594.333,A -85,B 0,C 180,E1 -19236.016,E2 -19236.016} C_VEL
LIN {X 0,Y 242.045,Z 594.335,A -85,B 0,C 180,E1 -19239.608,E2 -19239.608} C_VEL
LIN {X 0,Y 242.169,Z 594.319,A -85,B 0,C 180,E1 -19243.278,E2 -19243.278} C_VEL
LIN {X 0,Y 242.192,Z 594.318,A -85,B 0,C 180,E1 -19248.279,E2 -19248.279} C_VEL
LIN {X 0,Y 242.441,Z 594.284,A -85,B 0,C 180,E1 -19251.665,E2 -19251.665} C_VEL
LIN {X 0,Y 242.264,Z 594.306,A -85,B 0,C 180,E1 -19255.007,E2 -19255.007} C_VEL
LIN {X 0,Y 242.641,Z 594.262,A -85,B 0,C 180,E1 -19258.34,E2 -19258.34} C_VEL
LIN {X 0,Y 242.641,Z 594.256,A -85,B 0,C 180,E1 -19261.659,E2 -19261.659} C_VEL
LIN {X 0,Y 242.434,Z 594.28,A -85,B 0,C 180,E1 -19266.727,E2 -19266.727} C_VEL
LIN {X 0,Y 242.319,Z 594.3,A -85,B 0,C 180,E1 -19270.021,E2 -19270.021} C_VEL
LIN {X 0,Y 242.168,Z 594.307,A -85,B 0,C 180,E1 -19275.14,E2 -19275.14} C_VEL
LIN {X 0,Y 242.077,Z 594.328,A -85,B 0,C 180,E1 -19278.623,E2 -19278.623} C_VEL
LIN {X 0,Y 242.017,Z 594.339,A -85,B 0,C 180,E1 -19282.179,E2 -19282.179} C_VEL
LIN {X 0,Y 242.07,Z 594.323,A -85,B 0,C 180,E1 -19285.837,E2 -19285.837} C_VEL
LIN {X 0,Y 242.034,Z 594.332,A -85,B 0,C 180,E1 -19289.579,E2 -19289.579} C_VEL
LIN {X 0,Y 241.983,Z 594.339,A -85,B 0,C 180,E1 -19293.491,E2 -19293.491} C_VEL
LIN {X 0,Y 241.992,Z 594.339,A -85,B 0,C 180,E1 -19297.581,E2 -19297.581} C_VEL
LIN {X 0,Y 241.941,Z 594.346,A -85,B 0,C 180,E1 -19301.921,E2 -19301.921} C_VEL
LIN {X 0,Y 241.952,Z 594.342,A -85,B 0,C 180,E1 -19306.566,E2 -19306.566} C_VEL
LIN {X 0,Y 241.977,Z 594.343,A -85,B 0,C 180,E1 -19310.283,E2 -19310.283} C_VEL
LIN {X 0,Y 242.038,Z 594.335,A -85,B 0,C 180,E1 -19314.496,E2 -19314.496} C_VEL
LIN {X 0,Y 241.975,Z 594.34,A -85,B 0,C 180,E1 -19318.478,E2 -19318.478} C_VEL
LIN {X 0,Y 242.003,Z 594.34,A -85,B 0,C 180,E1 -19322.311,E2 -19322.311} C_VEL
LIN {X 0,Y 242.058,Z 594.333,A -85,B 0,C 180,E1 -19326.015,E2 -19326.015} C_VEL
LIN {X 0,Y 242.038,Z 594.334,A -85,B 0,C 180,E1 -19329.607,E2 -19329.607} C_VEL
LIN {X 0,Y 242.163,Z 594.317,A -85,B 0,C 180,E1 -19333.277,E2 -19333.277} C_VEL
LIN {X 0,Y 242.198,Z 594.312,A -85,B 0,C 180,E1 -19338.173,E2 -19338.173} C_VEL
LIN {X 0,Y 246.722,Z 606.887,A -85,B 0,C 180,E1 -19339.836,E2 -19339.836} C_VEL
LIN {X 0,Y 249.41,Z 616.167,A -85,B 0,C 180,E1 -19341.226,E2 -19341.226} C_VEL
LIN {X 0,Y 251.064,Z 623.568,A -85,B 0,C 180,E1 -19342.456,E2 -19342.456} C_VEL
LIN {X 0,Y 249.748,Z 633.848,A -85,B 0,C 180,E1 -19344.144,E2 -19344.144} C_VEL
LIN {X 0,Y 248.132,Z 644.522,A -85,B 0,C 180,E1 -19346.345,E2 -19346.345} C_VEL
LIN {X 0,Y 246.827,Z 652.428,A -85,B 0,C 180,E1 -19348.367,E2 -19348.367} C_VEL
LIN {X 0,Y 245.494,Z 660.192,A -85,B 0,C 180,E1 -19350.819,E2 -19350.819} C_VEL
LIN {X 0,Y 244.405,Z 666.42,A -85,B 0,C 180,E1 -19353.295,E2 -19353.295} C_VEL
LIN {X 0,Y 243.517,Z 671.404,A -85,B 0,C 180,E1 -19355.796,E2 -19355.796} C_VEL
LIN {X 0,Y 242.926,Z 675.268,A -85,B 0,C 180,E1 -19358.316,E2 -19358.316} C_VEL
LIN {X 0,Y 242.685,Z 677.342,A -85,B 0,C 180,E1 -19360.066,E2 -19360.066} C_VEL
LIN {X 0,Y 242.566,Z 678.865,A -85,B 0,C 180,E1 -19361.7,E2 -19361.7} C_VEL
LIN {X 0,Y 242.582,Z 679.995,A -85,B 0,C 180,E1 -19363.4,E2 -19363.4} C_VEL
LIN {X 0,Y 243.003,Z 681.079,A -85,B 0,C 180,E1 -19366.809,E2 -19366.809} C_VEL
LIN {X 0,Y 243.375,Z 681.015,A -85,B 0,C 180,E1 -19368.519,E2 -19368.519} C_VEL
LIN {X 0,Y 243.875,Z 680.517,A -85,B 0,C 180,E1 -19370.23,E2 -19370.23} C_VEL
LIN {X 0,Y 245.333,Z 678.378,A -85,B 0,C 180,E1 -19373.554,E2 -19373.554} C_VEL
LIN {X 0,Y 246.878,Z 675.451,A -85,B 0,C 180,E1 -19376.181,E2 -19376.181} C_VEL
LIN {X 0,Y 248.819,Z 671.16,A -85,B 0,C 180,E1 -19378.884,E2 -19378.884} C_VEL
LIN {X 0,Y 251.257,Z 665.256,A -85,B 0,C 180,E1 -19381.63,E2 -19381.63} C_VEL
LIN {X 0,Y 253.798,Z 658.356,A -85,B 0,C 180,E1 -19384.106,E2 -19384.106} C_VEL
LIN {X 0,Y 256.189,Z 651.184,A -85,B 0,C 180,E1 -19386.141,E2 -19386.141} C_VEL
LIN {X 0,Y 258.967,Z 641.485,A -85,B 0,C 180,E1 -19388.338,E2 -19388.338} C_VEL
LIN {X 0,Y 259.491,Z 638.562,A -85,B 0,C 180,E1 -19388.949,E2 -19388.949} C_VEL
LIN {X 0,Y 255.419,Z 633.109,A -85,B 0,C 180,E1 -19390.829,E2 -19390.829} C_VEL
LIN {X 0,Y 249.762,Z 627.403,A -85,B 0,C 180,E1 -19392.98,E2 -19392.98} C_VEL
LIN {X 0,Y 244.552,Z 622.199,A -85,B 0,C 180,E1 -19394.915,E2 -19394.915} C_VEL
LIN {X 0,Y 244.256,Z 621.485,A -85,B 0,C 180,E1 -19395.124,E2 -19395.124} C_VEL
LIN {X 0,Y 243.515,Z 630.05,A -85,B 0,C 180,E1 -19399.576,E2 -19399.576} C_VEL
LIN {X 0,Y 243.234,Z 634.888,A -85,B 0,C 180,E1 -19401.996,E2 -19401.996} C_VEL
LIN {X 0,Y 245.45,Z 648.223,A -85,B 0,C 180,E1 -19402.963,E2 -19402.963} C_VEL
LIN {X 0,Y 247.605,Z 662.386,A -85,B 0,C 180,E1 -19404.337,E2 -19404.337} C_VEL
LIN {X 0,Y 248.414,Z 667.475,A -85,B 0,C 180,E1 -19404.926,E2 -19404.926} C_VEL
LIN {X 0,Y 247.26,Z 679.018,A -85,B 0,C 180,E1 -19406.341,E2 -19406.341} C_VEL
LIN {X 0,Y 245.653,Z 691.61,A -85,B 0,C 180,E1 -19408.285,E2 -19408.285} C_VEL
LIN {X 0,Y 244.206,Z 702.111,A -85,B 0,C 180,E1 -19410.321,E2 -19410.321} C_VEL
LIN {X 0,Y 242.992,Z 711.053,A -85,B 0,C 180,E1 -19412.435,E2 -19412.435} C_VEL
LIN {X 0,Y 241.972,Z 718.749,A -85,B 0,C 180,E1 -19414.634,E2 -19414.634} C_VEL
LIN {X 0,Y 241.099,Z 726.255,A -85,B 0,C 180,E1 -19417.28,E2 -19417.28} C_VEL
LIN {X 0,Y 240.39,Z 733.074,A -85,B 0,C 180,E1 -19420.354,E2 -19420.354} C_VEL
LIN {X 0,Y 240.016,Z 737.467,A -85,B 0,C 180,E1 -19422.974,E2 -19422.974} C_VEL
LIN {X 0,Y 239.875,Z 740.286,A -85,B 0,C 180,E1 -19425.199,E2 -19425.199} C_VEL
LIN {X 0,Y 239.94,Z 742.931,A -85,B 0,C 180,E1 -19428.169,E2 -19428.169} C_VEL
LIN {X 0,Y 240.17,Z 743.848,A -85,B 0,C 180,E1 -19429.889,E2 -19429.889} C_VEL
LIN {X 0,Y 241.023,Z 744.489,A -85,B 0,C 180,E1 -19433.303,E2 -19433.303} C_VEL
LIN {X 0,Y 241.55,Z 744.196,A -85,B 0,C 180,E1 -19434.993,E2 -19434.993} C_VEL
LIN {X 0,Y 243.132,Z 742.418,A -85,B 0,C 180,E1 -19438.344,E2 -19438.344} C_VEL
LIN {X 0,Y 244.199,Z 740.945,A -85,B 0,C 180,E1 -19440.001,E2 -19440.001} C_VEL
LIN {X 0,Y 246.83,Z 736.699,A -85,B 0,C 180,E1 -19443.265,E2 -19443.265} C_VEL
LIN {X 0,Y 249.303,Z 732.359,A -85,B 0,C 180,E1 -19445.663,E2 -19445.663} C_VEL
LIN {X 0,Y 252.765,Z 725.845,A -85,B 0,C 180,E1 -19448.394,E2 -19448.394} C_VEL
LIN {X 0,Y 256.15,Z 718.905,A -85,B 0,C 180,E1 -19450.673,E2 -19450.673} C_VEL
LIN {X 0,Y 260.355,Z 709.547,A -85,B 0,C 180,E1 -19453.092,E2 -19453.092} C_VEL
LIN {X 0,Y 264.209,Z 699.945,A -85,B 0,C 180,E1 -19455.032,E2 -19455.032} C_VEL
LIN {X 0,Y 268.01,Z 689.381,A -85,B 0,C 180,E1 -19456.766,E2 -19456.766} C_VEL
LIN {X 0,Y 268.113,Z 682.245,A -85,B 0,C 180,E1 -19458.334,E2 -19458.334} C_VEL
LIN {X 0,Y 267.297,Z 673.679,A -85,B 0,C 180,E1 -19460.398,E2 -19460.398} C_VEL
LIN {X 0,Y 265.463,Z 663.952,A -85,B 0,C 180,E1 -19462.965,E2 -19462.965} C_VEL
LIN {X 0,Y 263.506,Z 656.25,A -85,B 0,C 180,E1 -19465.261,E2 -19465.261} C_VEL
LIN {X 0,Y 262.683,Z 653.245,A -85,B 0,C 180,E1 -19466.214,E2 -19466.214} C_VEL
LIN {X 0,Y 260.668,Z 648.405,A -85,B 0,C 180,E1 -19468.299,E2 -19468.299} C_VEL
LIN {X 0,Y 260.084,Z 647.58,A -85,B 0,C 180,E1 -19468.857,E2 -19468.857} C_VEL
LIN {X 0,Y 258.814,Z 646.392,A -85,B 0,C 180,E1 -19470.104,E2 -19470.104} C_VEL
LIN {X 0,Y 257.416,Z 646.232,A -85,B 0,C 180,E1 -19471.387,E2 -19471.387} C_VEL
LIN {X 0,Y 254.549,Z 647.17,A -85,B 0,C 180,E1 -19474.912,E2 -19474.912} C_VEL
LIN {X 0,Y 254.239,Z 646.931,A -85,B 0,C 180,E1 -19475.809,E2 -19475.809} C_VEL
LIN {X 0,Y 254.259,Z 646.092,A -85,B 0,C 180,E1 -19478.022,E2 -19478.022} C_VEL
LIN {X 0,Y 254.581,Z 646.306,A -85,B 0,C 180,E1 -19479.416,E2 -19479.416} C_VEL
LIN {X 0,Y 255.019,Z 647.547,A -85,B 0,C 180,E1 -19481.922,E2 -19481.922} C_VEL
LIN {X 0,Y 255.855,Z 650.064,A -85,B 0,C 180,E1 -19483.916,E2 -19483.916} C_VEL
LIN {X 0,Y 258.074,Z 655.169,A -85,B 0,C 180,E1 -19487.021,E2 -19487.021} C_VEL
LIN {X 0,Y 259.247,Z 660.725,A -85,B 0,C 180,E1 -19488.809,E2 -19488.809} C_VEL
LIN {X 0,Y 260.714,Z 672.609,A -85,B 0,C 180,E1 -19491.686,E2 -19491.686} C_VEL
LIN {X 0,Y 261.275,Z 682.822,A -85,B 0,C 180,E1 -19493.801,E2 -19493.801} C_VEL
LIN {X 0,Y 261.016,Z 693.496,A -85,B 0,C 180,E1 -19495.828,E2 -19495.828} C_VEL
LIN {X 0,Y 259.617,Z 703.97,A -85,B 0,C 180,E1 -19497.675,E2 -19497.675} C_VEL
LIN {X 0,Y 256.152,Z 716.113,A -85,B 0,C 180,E1 -19499.727,E2 -19499.727} C_VEL
LIN {X 0,Y 252.604,Z 726.373,A -85,B 0,C 180,E1 -19501.774,E2 -19501.774} C_VEL
LIN {X 0,Y 248.478,Z 735.982,A -85,B 0,C 180,E1 -19504,E2 -19504} C_VEL
LIN {X 0,Y 244.637,Z 743.993,A -85,B 0,C 180,E1 -19506.286,E2 -19506.286} C_VEL
LIN {X 0,Y 241.189,Z 751.038,A -85,B 0,C 180,E1 -19508.821,E2 -19508.821} C_VEL
LIN {X 0,Y 238.789,Z 756.165,A -85,B 0,C 180,E1 -19511.112,E2 -19511.112} C_VEL
LIN {X 0,Y 236.665,Z 760.637,A -85,B 0,C 180,E1 -19513.616,E2 -19513.616} C_VEL
LIN {X 0,Y 234.889,Z 764.147,A -85,B 0,C 180,E1 -19516.153,E2 -19516.153} C_VEL
LIN {X 0,Y 233.597,Z 767.441,A -85,B 0,C 180,E1 -19519.602,E2 -19519.602} C_VEL
LIN {X 0,Y 233.226,Z 768.52,A -85,B 0,C 180,E1 -19521.336,E2 -19521.336} C_VEL
LIN {X 0,Y 232.991,Z 769.46,A -85,B 0,C 180,E1 -19524.81,E2 -19524.81} C_VEL
LIN {X 0,Y 233.06,Z 769.347,A -85,B 0,C 180,E1 -19526.544,E2 -19526.544} C_VEL
LIN {X 0,Y 233.122,Z 768.836,A -85,B 0,C 180,E1 -19528.274,E2 -19528.274} C_VEL
LIN {X 0,Y 233.532,Z 767.922,A -85,B 0,C 180,E1 -19530.002,E2 -19530.002} C_VEL
LIN {X 0,Y 233.267,Z 766.482,A -85,B 0,C 180,E1 -19531.728,E2 -19531.728} C_VEL
LIN {X 0,Y 233.256,Z 763.517,A -85,B 0,C 180,E1 -19534.321,E2 -19534.321} C_VEL
LIN {X 0,Y 233.345,Z 759.421,A -85,B 0,C 180,E1 -19536.921,E2 -19536.921} C_VEL
LIN {X 0,Y 233.623,Z 753.045,A -85,B 0,C 180,E1 -19539.962,E2 -19539.962} C_VEL
LIN {X 0,Y 234.242,Z 745.983,A -85,B 0,C 180,E1 -19542.565,E2 -19542.565} C_VEL
LIN {X 0,Y 235.289,Z 737.237,A -85,B 0,C 180,E1 -19545.152,E2 -19545.152} C_VEL
LIN {X 0,Y 236.417,Z 728.268,A -85,B 0,C 180,E1 -19547.295,E2 -19547.295} C_VEL
LIN {X 0,Y 237.945,Z 717.302,A -85,B 0,C 180,E1 -19549.409,E2 -19549.409} C_VEL
LIN {X 0,Y 238.843,Z 710.848,A -85,B 0,C 180,E1 -19550.454,E2 -19550.454} C_VEL
LIN {X 0,Y 238.882,Z 699.413,A -85,B 0,C 180,E1 -19552.033,E2 -19552.033} C_VEL
LIN {X 0,Y 238.482,Z 683.403,A -85,B 0,C 180,E1 -19553.88,E2 -19553.88} C_VEL
LIN {X 0,Y 238.169,Z 670.621,A -85,B 0,C 180,E1 -19555.451,E2 -19555.451} C_VEL
LIN {X 0,Y 237.224,Z 657.315,A -85,B 0,C 180,E1 -19556.723,E2 -19556.723} C_VEL
LIN {X 0,Y 235.664,Z 642.964,A -85,B 0,C 180,E1 -19557.774,E2 -19557.774} C_VEL
LIN {X 0,Y 235.566,Z 636.341,A -85,B 0,C 180,E1 -19558.88,E2 -19558.88} C_VEL
LIN {X 0,Y 237.297,Z 625.779,A -85,B 0,C 180,E1 -19564.246,E2 -19564.246} C_VEL
LIN {X 0,Y 238.856,Z 618.202,A -85,B 0,C 180,E1 -19568.164,E2 -19568.164} C_VEL
LIN {X 0,Y 238.987,Z 616.487,A -85,B 0,C 180,E1 -19569.07,E2 -19569.07} C_VEL
LIN {X 0,Y 237.97,Z 610.573,A -85,B 0,C 180,E1 -19572.41,E2 -19572.41} C_VEL
LIN {X 0,Y 236.471,Z 603.104,A -85,B 0,C 180,E1 -19576.876,E2 -19576.876} C_VEL
LIN {X 0,Y 235.079,Z 595.686,A -85,B 0,C 180,E1 -19581.658,E2 -19581.658} C_VEL
LIN {X 0,Y 234.981,Z 595.223,A -85,B 0,C 180,E1 -19582.183,E2 -19582.183} C_VEL
LIN {X 0,Y 234.956,Z 595.223,A -85,B 0,C 180,E1 -19586.883,E2 -19586.883} C_VEL
LIN {X 0,Y 234.956,Z 595.217,A -85,B 0,C 180,E1 -19591.406,E2 -19591.406} C_VEL
LIN {X 0,Y 234.994,Z 595.212,A -85,B 0,C 180,E1 -19595.247,E2 -19595.247} C_VEL
LIN {X 0,Y 235.018,Z 595.211,A -85,B 0,C 180,E1 -19598.97,E2 -19598.97} C_VEL
LIN {X 0,Y 235.103,Z 595.2,A -85,B 0,C 180,E1 -19603.059,E2 -19603.059} C_VEL
LIN {X 0,Y 235.153,Z 595.194,A -85,B 0,C 180,E1 -19607.923,E2 -19607.923} C_VEL
LIN {X 0,Y 235.396,Z 595.161,A -85,B 0,C 180,E1 -19611.414,E2 -19611.414} C_VEL
LIN {X 0,Y 235.411,Z 595.16,A -85,B 0,C 180,E1 -19613.141,E2 -19613.141} C_VEL
LIN {X 0,Y 235.601,Z 595.138,A -85,B 0,C 180,E1 -19618.29,E2 -19618.29} C_VEL
LIN {X 0,Y 235.6,Z 595.133,A -85,B 0,C 180,E1 -19621.709,E2 -19621.709} C_VEL
LIN {X 0,Y 235.409,Z 595.156,A -85,B 0,C 180,E1 -19626.858,E2 -19626.858} C_VEL
LIN {X 0,Y 235.243,Z 595.183,A -85,B 0,C 180,E1 -19630.326,E2 -19630.326} C_VEL
LIN {X 0,Y 235.116,Z 595.184,A -85,B 0,C 180,E1 -19635.605,E2 -19635.605} C_VEL
LIN {X 0,Y 235.013,Z 595.207,A -85,B 0,C 180,E1 -19639.204,E2 -19639.204} C_VEL
LIN {X 0,Y 234.965,Z 595.214,A -85,B 0,C 180,E1 -19642.882,E2 -19642.882} C_VEL
LIN {X 0,Y 234.973,Z 595.204,A -85,B 0,C 180,E1 -19646.656,E2 -19646.656} C_VEL
LIN {X 0,Y 234.935,Z 595.222,A -85,B 0,C 180,E1 -19650.566,E2 -19650.566} C_VEL
LIN {X 0,Y 234.933,Z 595.221,A -85,B 0,C 180,E1 -19654.637,E2 -19654.637} C_VEL
LIN {X 0,Y 234.944,Z 595.217,A -85,B 0,C 180,E1 -19658.943,E2 -19658.943} C_VEL
LIN {X 0,Y 234.892,Z 595.219,A -85,B 0,C 180,E1 -19663.484,E2 -19663.484} C_VEL
LIN {X 0,Y 234.929,Z 595.216,A -85,B 0,C 180,E1 -19666.522,E2 -19666.522} C_VEL
LIN {X 0,Y 234.957,Z 595.211,A -85,B 0,C 180,E1 -19671.085,E2 -19671.085} C_VEL
LIN {X 0,Y 234.962,Z 595.215,A -85,B 0,C 180,E1 -19675.366,E2 -19675.366} C_VEL
LIN {X 0,Y 234.924,Z 595.219,A -85,B 0,C 180,E1 -19679.43,E2 -19679.43} C_VEL
LIN {X 0,Y 234.994,Z 595.209,A -85,B 0,C 180,E1 -19683.792,E2 -19683.792} C_VEL
LIN {X 0,Y 235.012,Z 595.211,A -85,B 0,C 180,E1 -19688.968,E2 -19688.968} C_VEL
LIN {X 0,Y 235.096,Z 595.198,A -85,B 0,C 180,E1 -19693.058,E2 -19693.058} C_VEL
LIN {X 0,Y 235.171,Z 595.387,A -85,B 0,C 180,E1 -19697.54,E2 -19697.54} C_VEL
LIN {X 0,Y 239.517,Z 607.255,A -85,B 0,C 180,E1 -19699.148,E2 -19699.148} C_VEL
LIN {X 0,Y 242.6,Z 617.386,A -85,B 0,C 180,E1 -19700.733,E2 -19700.733} C_VEL
LIN {X 0,Y 244.252,Z 625.594,A -85,B 0,C 180,E1 -19702.143,E2 -19702.143} C_VEL
LIN {X 0,Y 242.785,Z 636.187,A -85,B 0,C 180,E1 -19703.975,E2 -19703.975} C_VEL
LIN {X 0,Y 241.084,Z 646.652,A -85,B 0,C 180,E1 -19706.238,E2 -19706.238} C_VEL
LIN {X 0,Y 239.508,Z 655.599,A -85,B 0,C 180,E1 -19708.701,E2 -19708.701} C_VEL
LIN {X 0,Y 238.218,Z 663.026,A -85,B 0,C 180,E1 -19711.266,E2 -19711.266} C_VEL
LIN {X 0,Y 237.298,Z 668.013,A -85,B 0,C 180,E1 -19713.394,E2 -19713.394} C_VEL
LIN {X 0,Y 236.433,Z 672.875,A -85,B 0,C 180,E1 -19715.97,E2 -19715.97} C_VEL
LIN {X 0,Y 235.85,Z 676.63,A -85,B 0,C 180,E1 -19718.567,E2 -19718.567} C_VEL
LIN {X 0,Y 235.623,Z 678.586,A -85,B 0,C 180,E1 -19720.308,E2 -19720.308} C_VEL
LIN {X 0,Y 235.533,Z 680.077,A -85,B 0,C 180,E1 -19722.054,E2 -19722.054} C_VEL
LIN {X 0,Y 235.729,Z 681.843,A -85,B 0,C 180,E1 -19725.563,E2 -19725.563} C_VEL
LIN {X 0,Y 236.188,Z 682.105,A -85,B 0,C 180,E1 -19727.791,E2 -19727.791} C_VEL
LIN {X 0,Y 237.077,Z 681.423,A -85,B 0,C 180,E1 -19730.837,E2 -19730.837} C_VEL
LIN {X 0,Y 238.57,Z 679.337,A -85,B 0,C 180,E1 -19734.047,E2 -19734.047} C_VEL
LIN {X 0,Y 240.323,Z 676.095,A -85,B 0,C 180,E1 -19736.952,E2 -19736.952} C_VEL
LIN {X 0,Y 242.279,Z 672.006,A -85,B 0,C 180,E1 -19739.545,E2 -19739.545} C_VEL
LIN {X 0,Y 245,Z 665.645,A -85,B 0,C 180,E1 -19742.536,E2 -19742.536} C_VEL
LIN {X 0,Y 247.737,Z 658.533,A -85,B 0,C 180,E1 -19745.06,E2 -19745.06} C_VEL
LIN {X 0,Y 250.782,Z 649.511,A -85,B 0,C 180,E1 -19747.553,E2 -19747.553} C_VEL
LIN {X 0,Y 252.754,Z 642.89,A -85,B 0,C 180,E1 -19749.037,E2 -19749.037} C_VEL
LIN {X 0,Y 252.653,Z 641.146,A -85,B 0,C 180,E1 -19749.5,E2 -19749.5} C_VEL
LIN {X 0,Y 248.527,Z 636.101,A -85,B 0,C 180,E1 -19751.427,E2 -19751.427} C_VEL
LIN {X 0,Y 242.916,Z 630.654,A -85,B 0,C 180,E1 -19753.674,E2 -19753.674} C_VEL
LIN {X 0,Y 237.29,Z 625.269,A -85,B 0,C 180,E1 -19755.893,E2 -19755.893} C_VEL
LIN {X 0,Y 237.052,Z 624.697,A -85,B 0,C 180,E1 -19756.133,E2 -19756.133} C_VEL
LIN {X 0,Y 236.269,Z 634.566,A -85,B 0,C 180,E1 -19761.344,E2 -19761.344} C_VEL
LIN {X 0,Y 236.253,Z 635.059,A -85,B 0,C 180,E1 -19761.583,E2 -19761.583} C_VEL
LIN {X 0,Y 238.396,Z 648.541,A -85,B 0,C 180,E1 -19762.591,E2 -19762.591} C_VEL
LIN {X 0,Y 240.442,Z 661.905,A -85,B 0,C 180,E1 -19763.923,E2 -19763.923} C_VEL
LIN {X 0,Y 241.405,Z 669.403,A -85,B 0,C 180,E1 -19764.811,E2 -19764.811} C_VEL
LIN {X 0,Y 239.901,Z 681.798,A -85,B 0,C 180,E1 -19766.431,E2 -19766.431} C_VEL
LIN {X 0,Y 238.471,Z 693.018,A -85,B 0,C 180,E1 -19768.271,E2 -19768.271} C_VEL
LIN {X 0,Y 236.846,Z 704.758,A -85,B 0,C 180,E1 -19770.686,E2 -19770.686} C_VEL
LIN {X 0,Y 235.563,Z 713.581,A -85,B 0,C 180,E1 -19772.937,E2 -19772.937} C_VEL
LIN {X 0,Y 234.494,Z 722.196,A -85,B 0,C 180,E1 -19775.664,E2 -19775.664} C_VEL
LIN {X 0,Y 233.676,Z 729.066,A -85,B 0,C 180,E1 -19778.382,E2 -19778.382} C_VEL
LIN {X 0,Y 233.248,Z 733.678,A -85,B 0,C 180,E1 -19780.644,E2 -19780.644} C_VEL
LIN {X 0,Y 232.897,Z 738.033,A -85,B 0,C 180,E1 -19783.342,E2 -19783.342} C_VEL
LIN {X 0,Y 232.78,Z 741.252,A -85,B 0,C 180,E1 -19786.024,E2 -19786.024} C_VEL
LIN {X 0,Y 232.831,Z 742.807,A -85,B 0,C 180,E1 -19787.802,E2 -19787.802} C_VEL
LIN {X 0,Y 233.017,Z 743.947,A -85,B 0,C 180,E1 -19789.575,E2 -19789.575} C_VEL
LIN {X 0,Y 233.763,Z 744.962,A -85,B 0,C 180,E1 -19792.791,E2 -19792.791} C_VEL
LIN {X 0,Y 234.404,Z 744.87,A -85,B 0,C 180,E1 -19794.84,E2 -19794.84} C_VEL
LIN {X 0,Y 235.08,Z 744.398,A -85,B 0,C 180,E1 -19796.573,E2 -19796.573} C_VEL
LIN {X 0,Y 236.004,Z 743.515,A -85,B 0,C 180,E1 -19798.294,E2 -19798.294} C_VEL
LIN {X 0,Y 238.372,Z 740.546,A -85,B 0,C 180,E1 -19801.69,E2 -19801.69} C_VEL
LIN {X 0,Y 240.599,Z 737.238,A -85,B 0,C 180,E1 -19804.188,E2 -19804.188} C_VEL
LIN {X 0,Y 243.286,Z 732.906,A -85,B 0,C 180,E1 -19806.636,E2 -19806.636} C_VEL
LIN {X 0,Y 247.005,Z 726.5,A -85,B 0,C 180,E1 -19809.417,E2 -19809.417} C_VEL
LIN {X 0,Y 250.62,Z 719.576,A -85,B 0,C 180,E1 -19811.732,E2 -19811.732} C_VEL
LIN {X 0,Y 254.544,Z 711.512,A -85,B 0,C 180,E1 -19813.892,E2 -19813.892} C_VEL
LIN {X 0,Y 258.453,Z 702.747,A -85,B 0,C 180,E1 -19815.779,E2 -19815.779} C_VEL
LIN {X 0,Y 262.534,Z 692.2,A -85,B 0,C 180,E1 -19817.599,E2 -19817.599} C_VEL
LIN {X 0,Y 263.027,Z 687.376,A -85,B 0,C 180,E1 -19818.702,E2 -19818.702} C_VEL
LIN {X 0,Y 262.67,Z 678.356,A -85,B 0,C 180,E1 -19820.984,E2 -19820.984} C_VEL
LIN {X 0,Y 261.291,Z 668.117,A -85,B 0,C 180,E1 -19823.869,E2 -19823.869} C_VEL
LIN {X 0,Y 259.858,Z 661.133,A -85,B 0,C 180,E1 -19826.098,E2 -19826.098} C_VEL
LIN {X 0,Y 258.914,Z 657.514,A -85,B 0,C 180,E1 -19827.481,E2 -19827.481} C_VEL
LIN {X 0,Y 258.109,Z 654.882,A -85,B 0,C 180,E1 -19828.606,E2 -19828.606} C_VEL
LIN {X 0,Y 256.12,Z 650.478,A -85,B 0,C 180,E1 -19831.425,E2 -19831.425} C_VEL
LIN {X 0,Y 254.25,Z 646.987,A -85,B 0,C 180,E1 -19835.699,E2 -19835.699} C_VEL
LIN {X 0,Y 254.239,Z 646.931,A -85,B 0,C 180,E1 -19835.809,E2 -19835.809} C_VEL
LIN {X 0,Y 254.022,Z 647.004,A -85,B 0,C 180,E1 -19837.14,E2 -19837.14} C_VEL
LIN {X 0,Y 253.708,Z 648.239,A -85,B 0,C 180,E1 -19838.451,E2 -19838.451} C_VEL
LIN {X 0,Y 253.295,Z 655.446,A -85,B 0,C 180,E1 -19842.736,E2 -19842.736} C_VEL
LIN {X 0,Y 254.898,Z 660.091,A -85,B 0,C 180,E1 -19845.797,E2 -19845.797} C_VEL
LIN {X 0,Y 255.455,Z 661.49,A -85,B 0,C 180,E1 -19846.547,E2 -19846.547} C_VEL
LIN {X 0,Y 256.056,Z 666.403,A -85,B 0,C 180,E1 -19848.123,E2 -19848.123} C_VEL
LIN {X 0,Y 256.792,Z 677.753,A -85,B 0,C 180,E1 -19850.991,E2 -19850.991} C_VEL
LIN {X 0,Y 256.691,Z 688.976,A -85,B 0,C 180,E1 -19853.412,E2 -19853.412} C_VEL
LIN {X 0,Y 255.798,Z 698.486,A -85,B 0,C 180,E1 -19855.292,E2 -19855.292} C_VEL
LIN {X 0,Y 254.424,Z 706.023,A -85,B 0,C 180,E1 -19856.699,E2 -19856.699} C_VEL
LIN {X 0,Y 251.393,Z 715.589,A -85,B 0,C 180,E1 -19858.389,E2 -19858.389} C_VEL
LIN {X 0,Y 247.24,Z 726.603,A -85,B 0,C 180,E1 -19860.639,E2 -19860.639} C_VEL
LIN {X 0,Y 242.946,Z 735.969,A -85,B 0,C 180,E1 -19862.897,E2 -19862.897} C_VEL
LIN {X 0,Y 238.831,Z 743.819,A -85,B 0,C 180,E1 -19865.21,E2 -19865.21} C_VEL
LIN {X 0,Y 234.635,Z 751.826,A -85,B 0,C 180,E1 -19868.21,E2 -19868.21} C_VEL
LIN {X 0,Y 231.332,Z 758.141,A -85,B 0,C 180,E1 -19871.4,E2 -19871.4} C_VEL
LIN {X 0,Y 228.553,Z 763.224,A -85,B 0,C 180,E1 -19874.85,E2 -19874.85} C_VEL
LIN {X 0,Y 227.175,Z 765.933,A -85,B 0,C 180,E1 -19877.495,E2 -19877.495} C_VEL
LIN {X 0,Y 226.172,Z 768.21,A -85,B 0,C 180,E1 -19881.064,E2 -19881.064} C_VEL
LIN {X 0,Y 225.924,Z 768.975,A -85,B 0,C 180,E1 -19884.647,E2 -19884.647} C_VEL
LIN {X 0,Y 225.991,Z 768.787,A -85,B 0,C 180,E1 -19886.436,E2 -19886.436} C_VEL
LIN {X 0,Y 226.05,Z 768.16,A -85,B 0,C 180,E1 -19888.22,E2 -19888.22} C_VEL
LIN {X 0,Y 226.473,Z 767.14,A -85,B 0,C 180,E1 -19890.002,E2 -19890.002} C_VEL
LIN {X 0,Y 226.199,Z 765.621,A -85,B 0,C 180,E1 -19891.782,E2 -19891.782} C_VEL
LIN {X 0,Y 226.21,Z 762.492,A -85,B 0,C 180,E1 -19894.456,E2 -19894.456} C_VEL
LIN {X 0,Y 226.294,Z 758.22,A -85,B 0,C 180,E1 -19897.138,E2 -19897.138} C_VEL
LIN {X 0,Y 226.614,Z 751.604,A -85,B 0,C 180,E1 -19900.274,E2 -19900.274} C_VEL
LIN {X 0,Y 227.302,Z 744.379,A -85,B 0,C 180,E1 -19902.955,E2 -19902.955} C_VEL
LIN {X 0,Y 228.19,Z 737.024,A -85,B 0,C 180,E1 -19905.178,E2 -19905.178} C_VEL
LIN {X 0,Y 229.468,Z 727.104,A -85,B 0,C 180,E1 -19907.606,E2 -19907.606} C_VEL
LIN {X 0,Y 231.072,Z 716.023,A -85,B 0,C 180,E1 -19909.779,E2 -19909.779} C_VEL
LIN {X 0,Y 231.769,Z 709.304,A -85,B 0,C 180,E1 -19910.875,E2 -19910.875} C_VEL
LIN {X 0,Y 231.801,Z 697.639,A -85,B 0,C 180,E1 -19912.507,E2 -19912.507} C_VEL
LIN {X 0,Y 231.614,Z 686.499,A -85,B 0,C 180,E1 -19913.849,E2 -19913.849} C_VEL
LIN {X 0,Y 231.418,Z 675.375,A -85,B 0,C 180,E1 -19915.396,E2 -19915.396} C_VEL
LIN {X 0,Y 230.817,Z 662.694,A -85,B 0,C 180,E1 -19916.808,E2 -19916.808} C_VEL
LIN {X 0,Y 229.601,Z 649.044,A -85,B 0,C 180,E1 -19917.977,E2 -19917.977} C_VEL
LIN {X 0,Y 228.746,Z 641.512,A -85,B 0,C 180,E1 -19918.516,E2 -19918.516} C_VEL
LIN {X 0,Y 228.699,Z 635.282,A -85,B 0,C 180,E1 -19919.666,E2 -19919.666} C_VEL
LIN {X 0,Y 230.649,Z 624.447,A -85,B 0,C 180,E1 -19925.378,E2 -19925.378} C_VEL
LIN {X 0,Y 231.874,Z 618.345,A -85,B 0,C 180,E1 -19928.619,E2 -19928.619} C_VEL
LIN {X 0,Y 231.561,Z 614.823,A -85,B 0,C 180,E1 -19930.644,E2 -19930.644} C_VEL
LIN {X 0,Y 230.238,Z 608.233,A -85,B 0,C 180,E1 -19934.595,E2 -19934.595} C_VEL
LIN {X 0,Y 228.98,Z 601.739,A -85,B 0,C 180,E1 -19938.708,E2 -19938.708} C_VEL
LIN {X 0,Y 227.928,Z 596.102,A -85,B 0,C 180,E1 -19942.598,E2 -19942.598} C_VEL
LIN {X 0,Y 227.897,Z 596.104,A -85,B 0,C 180,E1 -19946.373,E2 -19946.373} C_VEL
LIN {X 0,Y 227.925,Z 596.095,A -85,B 0,C 180,E1 -19950.438,E2 -19950.438} C_VEL
LIN {X 0,Y 227.935,Z 596.094,A -85,B 0,C 180,E1 -19954.426,E2 -19954.426} C_VEL
LIN {X 0,Y 227.969,Z 596.09,A -85,B 0,C 180,E1 -19958.287,E2 -19958.287} C_VEL
LIN {X 0,Y 228.041,Z 596.081,A -85,B 0,C 180,E1 -19962.825,E2 -19962.825} C_VEL
LIN {X 0,Y 228.1,Z 596.071,A -85,B 0,C 180,E1 -19967.544,E2 -19967.544} C_VEL
LIN {X 0,Y 228.331,Z 596.042,A -85,B 0,C 180,E1 -19971.146,E2 -19971.146} C_VEL
LIN {X 0,Y 228.364,Z 596.038,A -85,B 0,C 180,E1 -19972.928,E2 -19972.928} C_VEL
LIN {X 0,Y 228.559,Z 596.015,A -85,B 0,C 180,E1 -19978.237,E2 -19978.237} C_VEL
LIN {X 0,Y 228.559,Z 596.011,A -85,B 0,C 180,E1 -19981.761,E2 -19981.761} C_VEL
LIN {X 0,Y 228.36,Z 596.033,A -85,B 0,C 180,E1 -19987.071,E2 -19987.071} C_VEL
LIN {X 0,Y 228.168,Z 596.063,A -85,B 0,C 180,E1 -19990.649,E2 -19990.649} C_VEL
LIN {X 0,Y 228.067,Z 596.067,A -85,B 0,C 180,E1 -19994.271,E2 -19994.271} C_VEL
LIN {X 0,Y 228.008,Z 596.074,A -85,B 0,C 180,E1 -19997.952,E2 -19997.952} C_VEL
LIN {X 0,Y 227.934,Z 596.094,A -85,B 0,C 180,E1 -20002.328,E2 -20002.328} C_VEL
LIN {X 0,Y 227.947,Z 596.079,A -85,B 0,C 180,E1 -20006.602,E2 -20006.602} C_VEL
LIN {X 0,Y 227.912,Z 596.094,A -85,B 0,C 180,E1 -20010.295,E2 -20010.295} C_VEL
LIN {X 0,Y 227.88,Z 596.096,A -85,B 0,C 180,E1 -20013.719,E2 -20013.719} C_VEL
LIN {X 0,Y 227.846,Z 596.102,A -85,B 0,C 180,E1 -20018.09,E2 -20018.09} C_VEL
LIN {X 0,Y 227.815,Z 596.103,A -85,B 0,C 180,E1 -20022.74,E2 -20022.74} C_VEL
LIN {X 0,Y 227.869,Z 596.097,A -85,B 0,C 180,E1 -20027.269,E2 -20027.269} C_VEL
LIN {X 0,Y 227.871,Z 596.093,A -85,B 0,C 180,E1 -20031.913,E2 -20031.913} C_VEL
LIN {X 0,Y 227.892,Z 596.098,A -85,B 0,C 180,E1 -20036.371,E2 -20036.371} C_VEL
LIN {X 0,Y 227.905,Z 596.097,A -85,B 0,C 180,E1 -20040.434,E2 -20040.434} C_VEL
LIN {X 0,Y 227.929,Z 596.092,A -85,B 0,C 180,E1 -20044.424,E2 -20044.424} C_VEL
LIN {X 0,Y 227.963,Z 596.088,A -85,B 0,C 180,E1 -20048.286,E2 -20048.286} C_VEL
LIN {X 0,Y 228.035,Z 596.079,A -85,B 0,C 180,E1 -20052.824,E2 -20052.824} C_VEL
LIN {X 0,Y 228.066,Z 596.077,A -85,B 0,C 180,E1 -20056.777,E2 -20056.777} C_VEL
LIN {X 0,Y 232.659,Z 608.588,A -85,B 0,C 180,E1 -20058.567,E2 -20058.567} C_VEL
LIN {X 0,Y 235.82,Z 618.82,A -85,B 0,C 180,E1 -20060.245,E2 -20060.245} C_VEL
LIN {X 0,Y 237.484,Z 626.943,A -85,B 0,C 180,E1 -20061.704,E2 -20061.704} C_VEL
LIN {X 0,Y 235.961,Z 637.477,A -85,B 0,C 180,E1 -20063.586,E2 -20063.586} C_VEL
LIN {X 0,Y 234.341,Z 647.019,A -85,B 0,C 180,E1 -20065.699,E2 -20065.699} C_VEL
LIN {X 0,Y 232.955,Z 654.846,A -85,B 0,C 180,E1 -20067.837,E2 -20067.837} C_VEL
LIN {X 0,Y 231.537,Z 662.511,A -85,B 0,C 180,E1 -20070.433,E2 -20070.433} C_VEL
LIN {X 0,Y 230.552,Z 667.775,A -85,B 0,C 180,E1 -20072.619,E2 -20072.619} C_VEL
LIN {X 0,Y 229.573,Z 672.902,A -85,B 0,C 180,E1 -20075.268,E2 -20075.268} C_VEL
LIN {X 0,Y 228.918,Z 676.896,A -85,B 0,C 180,E1 -20077.939,E2 -20077.939} C_VEL
LIN {X 0,Y 228.567,Z 679.863,A -85,B 0,C 180,E1 -20080.63,E2 -20080.63} C_VEL
LIN {X 0,Y 228.504,Z 681.282,A -85,B 0,C 180,E1 -20082.431,E2 -20082.431} C_VEL
LIN {X 0,Y 228.773,Z 682.95,A -85,B 0,C 180,E1 -20086.049,E2 -20086.049} C_VEL
LIN {X 0,Y 229.236,Z 683.124,A -85,B 0,C 180,E1 -20088.122,E2 -20088.122} C_VEL
LIN {X 0,Y 230.298,Z 682.331,A -85,B 0,C 180,E1 -20091.48,E2 -20091.48} C_VEL
LIN {X 0,Y 231.796,Z 680.311,A -85,B 0,C 180,E1 -20094.553,E2 -20094.553} C_VEL
LIN {X 0,Y 233.832,Z 676.734,A -85,B 0,C 180,E1 -20097.764,E2 -20097.764} C_VEL
LIN {X 0,Y 235.936,Z 672.524,A -85,B 0,C 180,E1 -20100.422,E2 -20100.422} C_VEL
LIN {X 0,Y 238.386,Z 667.043,A -85,B 0,C 180,E1 -20103.05,E2 -20103.05} C_VEL
LIN {X 0,Y 241.261,Z 660.066,A -85,B 0,C 180,E1 -20105.632,E2 -20105.632} C_VEL
LIN {X 0,Y 244.419,Z 651.159,A -85,B 0,C 180,E1 -20108.183,E2 -20108.183} C_VEL
LIN {X 0,Y 246.375,Z 644.996,A -85,B 0,C 180,E1 -20109.63,E2 -20109.63} C_VEL
LIN {X 0,Y 244.942,Z 642.708,A -85,B 0,C 180,E1 -20110.506,E2 -20110.506} C_VEL
LIN {X 0,Y 239.67,Z 637.356,A -85,B 0,C 180,E1 -20112.855,E2 -20112.855} C_VEL
LIN {X 0,Y 232.427,Z 630.493,A -85,B 0,C 180,E1 -20115.937,E2 -20115.937} C_VEL
LIN {X 0,Y 230.698,Z 629.37,A -85,B 0,C 180,E1 -20116.563,E2 -20116.563} C_VEL
LIN {X 0,Y 229.802,Z 627.894,A -85,B 0,C 180,E1 -20117.152,E2 -20117.152} C_VEL
LIN {X 0,Y 229.254,Z 635.353,A -85,B 0,C 180,E1 -20121.173,E2 -20121.173} C_VEL
LIN {X 0,Y 231.348,Z 648.374,A -85,B 0,C 180,E1 -20122.167,E2 -20122.167} C_VEL
LIN {X 0,Y 233.313,Z 661.556,A -85,B 0,C 180,E1 -20123.499,E2 -20123.499} C_VEL
LIN {X 0,Y 234.409,Z 668.863,A -85,B 0,C 180,E1 -20124.388,E2 -20124.388} C_VEL
LIN {X 0,Y 233.185,Z 680.034,A -85,B 0,C 180,E1 -20125.852,E2 -20125.852} C_VEL
LIN {X 0,Y 231.631,Z 691.658,A -85,B 0,C 180,E1 -20127.757,E2 -20127.757} C_VEL
LIN {X 0,Y 230.093,Z 702.608,A -85,B 0,C 180,E1 -20129.99,E2 -20129.99} C_VEL
LIN {X 0,Y 228.631,Z 712.698,A -85,B 0,C 180,E1 -20132.543,E2 -20132.543} C_VEL
LIN {X 0,Y 227.662,Z 720.245,A -85,B 0,C 180,E1 -20134.884,E2 -20134.884} C_VEL
LIN {X 0,Y 226.756,Z 727.566,A -85,B 0,C 180,E1 -20137.687,E2 -20137.687} C_VEL
LIN {X 0,Y 226.252,Z 732.533,A -85,B 0,C 180,E1 -20140.021,E2 -20140.021} C_VEL
LIN {X 0,Y 225.858,Z 737.266,A -85,B 0,C 180,E1 -20142.807,E2 -20142.807} C_VEL
LIN {X 0,Y 225.683,Z 740.807,A -85,B 0,C 180,E1 -20145.575,E2 -20145.575} C_VEL
LIN {X 0,Y 225.709,Z 742.595,A -85,B 0,C 180,E1 -20147.411,E2 -20147.411} C_VEL
LIN {X 0,Y 225.891,Z 743.946,A -85,B 0,C 180,E1 -20149.242,E2 -20149.242} C_VEL
LIN {X 0,Y 226.681,Z 745.362,A -85,B 0,C 180,E1 -20152.877,E2 -20152.877} C_VEL
LIN {X 0,Y 227.244,Z 745.488,A -85,B 0,C 180,E1 -20154.677,E2 -20154.677} C_VEL
LIN {X 0,Y 228.849,Z 744.512,A -85,B 0,C 180,E1 -20158.241,E2 -20158.241} C_VEL
LIN {X 0,Y 231.279,Z 742,A -85,B 0,C 180,E1 -20161.742,E2 -20161.742} C_VEL
LIN {X 0,Y 234.416,Z 737.83,A -85,B 0,C 180,E1 -20165.161,E2 -20165.161} C_VEL
LIN {X 0,Y 237.339,Z 733.56,A -85,B 0,C 180,E1 -20167.658,E2 -20167.658} C_VEL
LIN {X 0,Y 241.307,Z 727.184,A -85,B 0,C 180,E1 -20170.489,E2 -20170.489} C_VEL
LIN {X 0,Y 244.861,Z 721.067,A -85,B 0,C 180,E1 -20172.622,E2 -20172.622} C_VEL
LIN {X 0,Y 249.584,Z 712.032,A -85,B 0,C 180,E1 -20175.099,E2 -20175.099} C_VEL
LIN {X 0,Y 254.324,Z 701.887,A -85,B 0,C 180,E1 -20177.282,E2 -20177.282} C_VEL
LIN {X 0,Y 257.615,Z 693.91,A -85,B 0,C 180,E1 -20178.697,E2 -20178.697} C_VEL
LIN {X 0,Y 258.089,Z 686.085,A -85,B 0,C 180,E1 -20180.733,E2 -20180.733} C_VEL
LIN {X 0,Y 257.68,Z 677.672,A -85,B 0,C 180,E1 -20183.135,E2 -20183.135} C_VEL
LIN {X 0,Y 256.707,Z 668.691,A -85,B 0,C 180,E1 -20185.98,E2 -20185.98} C_VEL
LIN {X 0,Y 255.828,Z 663.764,A -85,B 0,C 180,E1 -20187.842,E2 -20187.842} C_VEL
LIN {X 0,Y 255.245,Z 661.297,A -85,B 0,C 180,E1 -20188.957,E2 -20188.957} C_VEL
LIN {X 0,Y 253.702,Z 656.989,A -85,B 0,C 180,E1 -20191.759,E2 -20191.759} C_VEL
LIN {X 0,Y 252.245,Z 653.556,A -85,B 0,C 180,E1 -20196.247,E2 -20196.247} C_VEL
